Universal Robots URScript: DAS428_958_02_MAR_21_DAS_lado_izquierdo_jig2.script

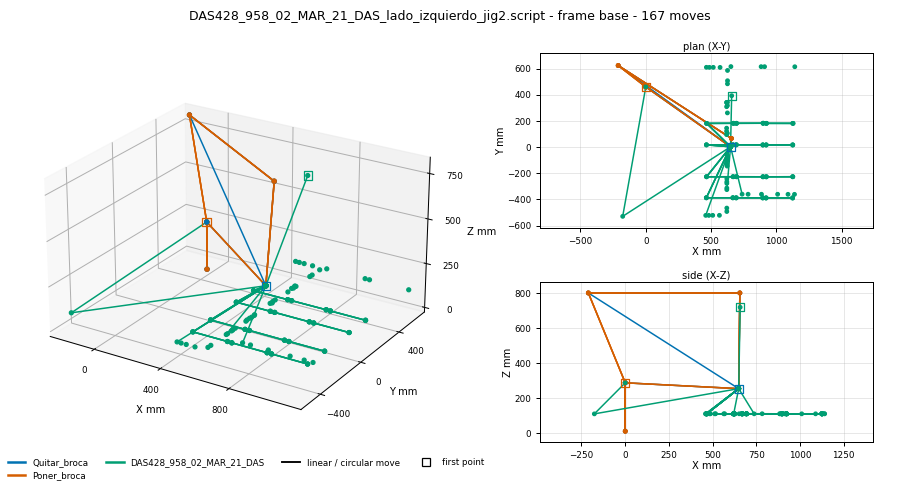
[picture p0: tool path of DAS428_958_02_MAR_21_DAS_lado_izquierdo_jig2.script in frame base, 167 of 755 moves have a stored position in this frame; points joined in program order, loops and branches not executed]
def DAS428_958_02_MAR_21_DAS_lado_izquierdo_jig2():
  step_count_cb486e1e_2b8d_495c_afa4_48e8c6bfd957 = 0
  thread Step_Counter_Thread_418e8cb4_311f_44ce_a52e_b6628405cc57():
    while (True):
      step_count_cb486e1e_2b8d_495c_afa4_48e8c6bfd957 = step_count_cb486e1e_2b8d_495c_afa4_48e8c6bfd957 + 1
      sync()
    end
  end
  run Step_Counter_Thread_418e8cb4_311f_44ce_a52e_b6628405cc57()
  set_safety_mode_transition_hardness(1)
  set_tcp(p[4.109330471764039E-4,-0.21829828276152607,0.037994196120996,1.5580092985761962,-0.12546870791316503,0.12120248426608284])
  set_payload(1.5)
  modbus_add_signal("192.168.10.45", 255, 187, 1, "postrnas_m187", False)
  modbus_set_signal_update_frequency("postrnas_m187", 10)
  modbus_add_signal("192.168.10.45", 255, 289, 1, "ini_cambro_m289", False)
  modbus_set_signal_update_frequency("ini_cambro_m289", 10)
  modbus_add_signal("192.168.10.45", 255, 290, 0, "fin_cambro_m290", False)
  modbus_set_signal_update_frequency("fin_cambro_m290", 10)
  modbus_add_signal("192.168.10.45", 255, 291, 1, "outputbroc_m291", False)
  modbus_set_signal_update_frequency("outputbroc_m291", 10)
  modbus_add_signal("192.168.10.45", 255, 292, 0, "fciclocarr_m292", False)
  modbus_set_signal_update_frequency("fciclocarr_m292", 10)
  modbus_add_signal("192.168.10.45", 255, 7, 1, "avancarrusel_m7", False)
  modbus_set_signal_update_frequency("avancarrusel_m7", 10)
  modbus_add_signal("192.168.10.45", 255, 252, 1, "pose2_m252", False)
  modbus_set_signal_update_frequency("pose2_m252", 10)
  modbus_add_signal("192.168.10.45", 255, 253, 1, "pose3_m253", False)
  modbus_set_signal_update_frequency("pose3_m253", 10)
  modbus_add_signal("192.168.10.45", 255, 254, 1, "pose4_m254", False)
  modbus_set_signal_update_frequency("pose4_m254", 10)
  modbus_add_signal("192.168.10.45", 255, 441, 1, "finciclo_m441", False)
  modbus_set_signal_update_frequency("finciclo_m441", 10)
  modbus_add_signal("192.168.10.45", 255, 442, 1, "finciclo_m442", False)
  modbus_set_signal_update_frequency("finciclo_m442", 10)
  modbus_add_signal("192.168.10.45", 255, 443, 1, "finciclo_m443", False)
  modbus_set_signal_update_frequency("finciclo_m443", 10)
  modbus_add_signal("192.168.10.45", 255, 503, 0, "homecobot_m503", False)
  modbus_set_signal_update_frequency("homecobot_m503", 10)
  modbus_add_signal("192.168.10.45", 255, 288, 1, "cargar_run_m288", False)
  modbus_set_signal_update_frequency("cargar_run_m288", 10)
  modbus_add_signal("192.168.10.45", 255, 287, 0, "desactiver_m288", False)
  modbus_set_signal_update_frequency("desactiver_m288", 10)
  modbus_add_signal("192.168.10.45", 255, 183, 0, "eje7home_m183", False)
  modbus_set_signal_update_frequency("eje7home_m183", 10)
  modbus_add_signal("192.168.10.45", 255, 444, 1, "finciclo_m444", False)
  modbus_set_signal_update_frequency("finciclo_m444", 10)
  modbus_add_signal("192.168.10.45", 255, 381, 0, "pat1_m381", False)
  modbus_set_signal_update_frequency("pat1_m381", 10)
  modbus_add_signal("192.168.10.45", 255, 382, 0, "pat2_m382", False)
  modbus_set_signal_update_frequency("pat2_m382", 10)
  modbus_add_signal("192.168.10.45", 255, 383, 0, "pat3_m383", False)
  modbus_set_signal_update_frequency("pat3_m383", 10)
  modbus_add_signal("192.168.10.45", 255, 384, 0, "pat4_m384", False)
  modbus_set_signal_update_frequency("pat4_m384", 10)
  modbus_add_signal("192.168.10.45", 255, 385, 0, "pat5_m385", False)
  modbus_set_signal_update_frequency("pat5_m385", 10)
  modbus_add_signal("192.168.10.45", 255, 386, 0, "pat6_m386", False)
  modbus_set_signal_update_frequency("pat6_m386", 10)
  modbus_add_signal("192.168.10.45", 255, 387, 0, "pat7_m387", False)
  modbus_set_signal_update_frequency("pat7_m387", 10)
  modbus_add_signal("192.168.10.45", 255, 388, 0, "pat8_m388", False)
  modbus_set_signal_update_frequency("pat8_m388", 10)
  modbus_add_signal("192.168.10.45", 255, 389, 0, "pat9_m389", False)
  modbus_set_signal_update_frequency("pat9_m389", 10)
  modbus_add_signal("192.168.10.45", 255, 390, 0, "pat10_m390", False)
  modbus_set_signal_update_frequency("pat10_m390", 10)
  modbus_add_signal("192.168.10.45", 255, 391, 0, "pat11_m391", False)
  modbus_set_signal_update_frequency("pat11_m391", 10)
  modbus_add_signal("192.168.10.45", 255, 392, 0, "pat12_m392", False)
  modbus_set_signal_update_frequency("pat12_m392", 10)
  modbus_add_signal("192.168.10.45", 255, 401, 0, "inipat1_m401", False)
  modbus_set_signal_update_frequency("inipat1_m401", 10)
  modbus_add_signal("192.168.10.45", 255, 402, 0, "inipat2_m402", False)
  modbus_set_signal_update_frequency("inipat2_m402", 10)
  modbus_add_signal("192.168.10.45", 255, 403, 0, "inipat3_m403", False)
  modbus_set_signal_update_frequency("inipat3_m403", 10)
  modbus_add_signal("192.168.10.45", 255, 404, 0, "inipat4_m404", False)
  modbus_set_signal_update_frequency("inipat4_m404", 10)
  modbus_add_signal("192.168.10.45", 255, 405, 0, "inipat5_m405", False)
  modbus_set_signal_update_frequency("inipat5_m405", 10)
  modbus_add_signal("192.168.10.45", 255, 406, 0, "inipat6_m406", False)
  modbus_set_signal_update_frequency("inipat6_m406", 10)
  modbus_add_signal("192.168.10.45", 255, 407, 0, "inipat7_m407", False)
  modbus_set_signal_update_frequency("inipat7_m407", 10)
  modbus_add_signal("192.168.10.45", 255, 408, 0, "inipat8_m408", False)
  modbus_set_signal_update_frequency("inipat8_m408", 10)
  modbus_add_signal("192.168.10.45", 255, 409, 0, "inipat9_m409", False)
  modbus_set_signal_update_frequency("inipat9_m409", 10)
  modbus_add_signal("192.168.10.45", 255, 410, 0, "inipat10_m410", False)
  modbus_set_signal_update_frequency("inipat10_m410", 10)
  modbus_add_signal("192.168.10.45", 255, 411, 0, "inipat11_m411", False)
  modbus_set_signal_update_frequency("inipat11_m411", 10)
  modbus_add_signal("192.168.10.45", 255, 412, 0, "inipat12_m412", False)
  modbus_set_signal_update_frequency("inipat12_m412", 10)
  modbus_add_signal("192.168.10.45", 255, 430, 0, "modeloDer_m430", False)
  modbus_set_signal_update_frequency("modeloDer_m430", 10)
  modbus_add_signal("192.168.10.45", 255, 380, 1, "mensaje_m380", False)
  modbus_set_signal_update_frequency("mensaje_m380", 10)
  modbus_add_signal("192.168.10.45", 255, 379, 0, "respues_m379", False)
  modbus_set_signal_update_frequency("respues_m379", 10)
  modbus_add_signal("192.168.10.45", 255, 251, 1, "pose1_m251", False)
  modbus_set_signal_update_frequency("pose1_m251", 10)
  modbus_set_runstate_dependent_choice("postrnas_m187",0)
  modbus_set_runstate_dependent_choice("ini_cambro_m289",0)
  modbus_set_runstate_dependent_choice("outputbroc_m291",0)
  modbus_set_runstate_dependent_choice("avancarrusel_m7",0)
  modbus_set_runstate_dependent_choice("pose2_m252",0)
  modbus_set_runstate_dependent_choice("pose3_m253",0)
  modbus_set_runstate_dependent_choice("pose4_m254",0)
  modbus_set_runstate_dependent_choice("finciclo_m441",0)
  modbus_set_runstate_dependent_choice("finciclo_m442",0)
  modbus_set_runstate_dependent_choice("finciclo_m443",0)
  modbus_set_runstate_dependent_choice("cargar_run_m288",0)
  modbus_set_runstate_dependent_choice("finciclo_m444",0)
  modbus_set_runstate_dependent_choice("mensaje_m380",0)
  modbus_set_runstate_dependent_choice("pose1_m251",0)
  set_standard_analog_input_domain(0, 1)
  set_standard_analog_input_domain(1, 1)
  set_tool_analog_input_domain(0, 1)
  set_tool_analog_input_domain(1, 1)
  set_analog_outputdomain(0, 0)
  set_analog_outputdomain(1, 0)
  set_input_actions_to_default()
  set_runstate_standard_digital_outputs([2])
  set_runstate_configurable_digital_outputs([1])
  set_runstate_standard_digital_output_to_value(2, 1)
  set_runstate_configurable_digital_output_to_value(1, 1)
  set_gravity([0.0, 0.0, 9.82])
  set_tool_communication(False, 115200, 0, 1, 1.5, 3.5)
  set_tool_output_mode(0)
  set_tool_digital_output_mode(0, 1)
  set_tool_digital_output_mode(1, 1)
  set_tool_voltage(0)
  global contador=0
  global i_var_1=0
  global Pallet_1_cnt_1=1
  global Pallet_1_cnt=1
  global Line_1=p[0.0,0.0,0.0,0.0,0.0,0.0]
  global Line_2=p[0.0,0.0,0.0,0.0,0.0,0.0]
  global Line_3=p[0.0,0.0,0.0,0.0,0.0,0.0]
  global Line_4=p[-0.2932874787951964,0.3932288129452105,0.013749459185886714,0.019478391032120013,-0.0350876085014595,1.5300278925331599]
  global Line_5=p[0.0,0.0,0.0,0.0,0.0,0.0]
  global Plane_1=p[-0.4357649673792705,0.3571224276764373,-0.011331751409534768,-0.03455953496512708,-0.012487423981114925,3.103751116092306]
  global Plane_2=p[-0.4823864034329737,0.3302516442079689,0.014283714098506706,0.017125077458443067,0.05770060098903715,-2.9134709732588786]
  global Plane_3=p[0.003678615545088639,0.4082921331082374,0.10477407557236007,-2.072177303174012E-4,7.379081343290108E-4,-6.424400645467977E-4]
  global Plane_4=p[-0.4500206307677429,-0.2823718146925442,-0.4767416657426552,0.013278190059218174,0.013334473770785706,1.8479691991032237]
  global Plano_patron1=p[-0.7699005610122596,0.304894434078545,0.0420369514744936,-0.0031270356010209216,1.7180543614697593E-4,-3.508888786211572E-5]
  global Point_13=p[0.0,0.0,0.0,0.0,0.0,0.0]
  global Point_3=p[0.0,0.0,0.0,0.0,0.0,0.0]
  global Point_8=p[0.0,0.0,0.0,0.0,0.0,0.0]
  global Punto_prot_1=p[0.0,0.0,0.0,0.0,0.0,0.0]
  global Punto_seg_der=p[0.23741638234469645,0.3587772222537799,0.42419077585740217,0.818517054876345,1.4216436941132238,1.005041187710707]
  global pisp_958=p[-0.41395442210486977,-0.2082168853247176,0.041553466664982,0.014014788518713659,0.01101911827984854,1.569193423241601]
  rtde_set_watchdog("speed_slider_mask", 10.0, "ignore")
  global Traslacion_p=p[.657998712498, .394119076430, .719668538659, .745859698144, 2.906519637838, .095468097993]
  global Traslacion_q=[-3.020863008919047, -1.4521287285823696, 0.9893999609737083, 0.3161356049923509, -5.817383157179211, 7.125860208047008E-4]
  global Home2_p=p[.649602302195, .003200282484, .254149874925, -2.448457879294, -1.966199736652, -.011076409707]
  global Home2_q=[-3.47968947108801, -1.6856169348881274, 2.036329601799979, -0.3455951480915882, -4.992365550646321, 0.0060764790449239214]
  global Home3_p=p[.649602302195, .003200282484, .254149874925, -2.448457879294, -1.966199736652, -.011076409707]
  global Home3_q=[-3.479689471087993, -1.6856169348881211, 2.0363296017999737, -0.34559514809159, -4.992365550646304, 0.006076479044924019]
  global Home4_p=p[.649602302195, .003200282484, .254149874925, -2.448457879294, -1.966199736652, -.011076409707]
  global Home4_q=[-3.479689471087993, -1.6856169348881211, 2.0363296017999737, -0.34559514809159, -4.992365550646304, 0.006076479044924019]
  global PosicionApagado_p=p[-.175961014487, -.529389253007, .109949884724, .175001600804, 2.113291246609, -2.157399109703]
  global PosicionApagado_q=[-1.5727354621284952, -1.5704867605983486, -2.807039864148308, -0.30557696332673245, -4.706711136129834, 1.778107977035495E-5]
  global Precambio_broca_p=p[.000830370305, .461517540512, .287521124194, -.221784750204, -3.131955254916, .000429460883]
  global Precambio_broca_q=[-2.1838225298159477, -2.0964618902985066, 2.243453456263678, -0.13436505871461257, -5.342774534909408, -0.004043449473680738]
  global Linea1_A_p=p[.465780239716, -.226284822275, .110110305320, 3.129199777247, .273979671894, -.008474561279]
  global Linea1_A_q=[-3.7622293747396913, -1.6873556925995992, 2.323362421011069, -0.625104012809361, -4.0968533396839515, 0.0033473062041684543]
  global Linea1_B_p=p[.669199999133, -.226066231601, .110221514703, 3.129199488643, .274057096186, -.008522317905]
  global Linea1_B_q=[-3.557231781452517, -1.3492008498278363, 1.961545229349972, -0.5993084840575982, -3.891978745553196, 0.0068914536813957416]
  global Linea1_C_p=p[.694599999674, -.226083076366, .110775282131, 3.129206209142, .274048762949, -.008557115599]
  global Linea1_C_q=[-3.5408294989047437, -1.3120520197143488, 1.9116878668393618, -0.5863558735051146, -3.8755559725861075, 0.007215554028316085]
  global Linea1_D_p=p[.897799999597, -.226330598752, .110549197198, 3.129164560911, .274100632214, -.008493112790]
  global Linea1_D_q=[-3.4452506974721455, -1.015094527261077, 1.4697422225132426, -0.4398923161705586, -3.779757131526884, 0.009316440733303288]
  global Linea1_E_p=p[.923199997743, -.226496087218, .110278761023, 3.129196935269, .274071665669, -.008639622731]
  global Linea1_E_q=[-3.436588597727809, -0.976349509057826, 1.4065148117166615, -0.4151627604596042, -3.7710218003171097, 0.009513196103198673]
  global Linea1_F_p=p[1.125593354651, -.226031138561, .110601831768, 3.129192254502, .274074519951, -.008696700454]
  global Linea1_F_q=[-3.380697676481182, -0.6099111929302072, 0.7528298757650722, -0.1267902515679964, -3.714400713814072, 0.010912064972982147]
  def calculate_point_to_move_towards(feature, direction, position_distance):
    local posDir=[direction[0], direction[1], direction[2]]
    if (norm(posDir) < 1e-6):
      return get_target_waypoint()
    end
    local direction_vector_normalized=normalize(posDir)
    local displacement_pose=p[direction_vector_normalized[0] * position_distance,direction_vector_normalized[1] * position_distance,direction_vector_normalized[2] * position_distance,0,0,0]
    local wanted_displacement_in_base_frame=pose_sub(pose_trans(feature, displacement_pose), feature)
    return pose_add(get_target_waypoint(), wanted_displacement_in_base_frame)
  end
  global Linea2_A_p=p[.466954168710, .182156727796, .110171699464, -2.448457838983, -1.966199888042, -.011076390033]
  global Linea2_A_q=[-3.096264362332022, -1.8105063261906196, 2.419381749575411, -0.604569943120544, -4.609367858418758, 0.008210447251383535]
  global Linea2_B_p=p[.671809999536, .182878038708, .110175282179, -2.448398718020, -1.966214966670, -.010953917198]
  global Linea2_B_q=[-3.112193266343249, -1.4618930385561022, 2.1005475692711357, -0.6342202128720773, -4.625507134533515, 0.00845567105716949]
  global Linea2_C_p=p[.694980620228, .182769618296, .110459932861, -2.448327792652, -1.966241960778, -.010898882344]
  global Linea2_C_q=[-3.1136170783763246, -1.427697328825201, 2.059986020915073, -0.6277999413035573, -4.626970277725095, 0.008475304624878617]
  global Linea2_D_p=p[.898787430028, .183234989861, .110403286316, -2.448304893977, -1.966353718915, -.010975641562]
  global Linea2_D_q=[-3.12042574519119, -1.1376151787135544, 1.6647315225706083, -0.5226894752077342, -4.633689721395611, 0.008491290355203619]
  global Linea2_E_p=p[.923789841802, .182506729307, .110323521287, -2.448339335785, -1.966352412105, -.011034134800]
  global Linea2_E_q=[-3.1220303350773233, -1.1024169697310633, 1.610792612077442, -0.5039930836645397, -4.635244042411777, 0.008484609097352974]
  global Linea2_F_p=p[1.126945944045, .182371421241, .110084235246, -2.448292218177, -1.966366471653, -.011020014588]
  global Linea2_F_q=[-3.126205891145389, -0.7888654762746627, 1.0844527378197477, -0.2911805586510319, -4.6389576225939395, 0.008426573530911268]
  global Linea7_A_p=p[.737913382913, -.359696656416, .110246852616, 3.131872092311, .186635383423, -.000389334829]
  global Linea7_A_q=[-3.681156562266171, -1.1996168071622932, 1.757330151202673, -0.5522026597660465, -3.9601640674441323, 0.005316316519943243]
  global Linea7_B_p=p[.783713148217, -.360080715325, .110620974020, 3.131872080694, .186635404395, -.000389343545]
  global Linea7_B_q=[-3.650143104990655, -1.1359413316685298, 1.6616529669860118, -0.5200665751996176, -3.929093763815281, 0.005555397450602444]
  global Linea8_A_p=p[.886282799932, -.360229310841, .110453772921, 3.131519956407, .186494776915, .000579777937]
  global Linea8_A_q=[-3.591304287493482, -0.9891617182428476, 1.4289624761138866, -0.4346002764061705, -3.870006358141346, 0.006011745682200086]
  global Linea8_B_p=p[1.009987450255, -.360229310302, .110179227584, 3.131519925151, .186494817820, .000579759973]
  global Linea8_B_q=[-3.5358660704998717, -0.7924298121308935, 1.0907006839592273, -0.2928265782260997, -3.8142305776877343, 0.0064076248760271785]
  global Linea9_A_p=p[1.089313325367, -.360630550626, .110237381886, 3.131274831042, .186572958872, .001401500331]
  global Linea9_A_q=[-3.507282006423159, -0.6385942191612735, 0.8089501351297868, -0.1653539889318978, -3.785363860326909, 0.006616479785108709]
  global Linea9_B_p=p[1.138944388844, -.360869351507, .110826017632, 3.131274802661, .186572988174, .001401483023]
  global Linea9_B_q=[-3.4914339632991864, -0.5124624399707418, 0.5676507222077732, -0.05011131989687101, -3.7691835676211607, 0.006732071657192494]
  global Linea10_A_p=p[.620978322043, -.324892456797, .110623766440, 3.127402623628, -.245143091263, -.004063554207]
  global Linea10_A_q=[-3.6869382053447044, -1.3223584773988293, 1.927375204305715, -0.5983630349819116, -3.6905142249820324, 0.0056231827538635315]
  global Linea10_B_p=p[.621097917225, -.276980216964, .110320290981, 3.127402605879, -.245143081258, -.004063559866]
  global Linea10_B_q=[-3.6188087722380935, -1.3384072237024949, 1.949063614559142, -0.6032315503323895, -3.6223937108691318, 0.006590396406481958]
  global Linea11_A_p=p[.623455356385, -.144672989900, .110191487849, -2.632012907887, -1.710466693368, -.008551801775]
  global Linea11_A_q=[-3.7294766647125748, -1.5700524659119814, 2.21580175367518, -0.6379282889546607, -5.042121691434226, 0.005581533742989642]
  global Linea11_B_p=p[.624119671393, -.090095469021, .110353884155, -2.632012896780, -1.710466734062, -.008551794970]
  global Linea11_B_q=[-3.6247502966617073, -1.585150048761757, 2.2304099707796063, -0.6377871669514974, -4.937393005511421, 0.006400309223622675]
  global Linea12_A_p=p[.624141411120, -.066274166300, .110334660294, -2.632061457031, -1.710628419892, -.008680091079]
  global Linea12_A_q=[-3.576867818672329, -1.5888248455929554, 2.23409769230859, -0.638081681915871, -4.88958008805711, 0.006759858484637715]
  global Linea12_B_p=p[.625005135416, .106664404916, .110180545519, -2.632061469151, -1.710628482598, -.008680127081]
  global Linea12_B_q=[-3.2068887547507323, -1.551909790420524, 2.1974871560020848, -0.638805025446775, -4.519623607927026, 0.009359012311380255]
  global Linea13_A_p=p[.625493298354, .262478777538, .110355483985, -2.632548083396, -1.710921113652, -.010070841951]
  global Linea13_A_q=[-2.896364151370071, -1.4448052024132805, 2.0799552622917368, -0.6290694071523859, -4.209104057924403, 0.011452105368751556]
  global Linea13_B_p=p[.625493296860, .318856578939, .110131630173, -2.632548086986, -1.710921163442, -.010070846484]
  global Linea13_B_q=[-2.7987199569733097, -1.394849229494266, 2.020507255629248, -0.6192929302058419, -4.111456896339345, 0.012194173917594142]
  global Linea14_A_p=p[.625748762392, .343504937265, .110090990642, -2.632595117185, -1.711060508708, -.011002715073]
  global Linea14_A_q=[-2.7589776121724974, -1.371725061704466, 1.991938508379024, -0.614306407879349, -4.0717686455064666, 0.012519321582973785]
  global Linea14_B_p=p[.626022539964, .485152545421, .110593753972, -2.632595124419, -1.711060553733, -.011002727305]
  global Linea14_B_q=[-2.561324434207597, -1.228184115147677, 1.79766140697026, -0.5625917279677406, -3.874049521809336, 0.014268843198803616]
  global Linea15_A_p=p[.626306650398, .508674603028, .110445455669, -2.632595127775, -1.711060613121, -.011002737975]
  global Linea15_A_q=[-2.533508862703878, -1.202261171286347, 1.7605999966793635, -0.55125669711577, -3.846216171124823, 0.014567785906905393]
  global Linea15_B_p=p[.626327608491, .587415564298, .110050045410, -2.632661246672, -1.711049389617, -.010999857798]
  global Linea15_B_q=[-2.4482942280068585, -1.1131828351876312, 1.6277564152308788, -0.5068229975694187, -3.760894753760676, 0.015518000293985423]
  global Linea16_A_p=p[.464714302335, .611413139504, .110697464349, -1.544268383540, -2.732104823202, -.006884184964]
  global Linea16_A_q=[-2.4550359831168613, -1.3587121352385232, 1.9739909556549193, -0.6095013542703764, -4.727784672200272, 0.006868741264362654]
  global Linea16_B_p=p[.487741348141, .611017673565, .110415464036, -1.544268358835, -2.732104854917, -.006884177480]
  global Linea16_B_q=[-2.4794279049425754, -1.3389262434910556, 1.9490984118290324, -0.604365353535707, -4.75217062245783, 0.006734800587170575]
  global Linea17_A_p=p[.517383659268, .611103429132, .110729179233, -1.544779713402, -2.732685367780, -.009945500495]
  global Linea17_A_q=[-2.5082575279683113, -1.3131453182243042, 1.9151753969774692, -0.598283135183288, -4.78088650060061, 0.00668272054728547]
  global Linea17_B_p=p[.569253413106, .610696887479, .110460451666, -1.544779672167, -2.732685417131, -.009945491911]
  global Linea17_B_q=[-2.5549019817458243, -1.2642731579102362, 1.8492778264267276, -0.5811941707445918, -4.827506542897114, 0.006516537786687767]
  global Linea18_A_p=p[.652275282871, .616966070789, .110402012202, -1.544268371887, -2.732104838867, -.006884188160]
  global Linea18_A_q=[-2.6106362750002035, -1.1730578134725853, 1.7176129055392177, -0.5385325271143078, -4.883275143872667, 0.005979356975084116]
  global Linea18_AB_p=p[.883614943259, .616349563116, .110351134256, -1.544268345639, -2.732104870876, -.006884192709]
  global Linea18_AB_q=[-2.7386992398245744, -0.9017900558849279, 1.281606576558123, -0.3734626609773617, -5.010988146234565, 0.005130637771908034]
  global Linea18_BA_p=p[.909904961943, .616222280799, .110421447666, -1.544268322161, -2.732104902209, -.006884182125]
  global Linea18_BA_q=[-2.7498726987223208, -0.8660697617883866, 1.2197485096371476, -0.3472882558118906, -5.02209865790525, 0.005047885057257062]
  global Linea18_B_p=p[1.141235285063, .615792039333, .110307833561, -1.544268303833, -2.732104945128, -.006884144817]
  global Linea18_B_q=[-2.8277732907081354, -0.39061700846990277, 0.32871463965525227, 0.06857809871196263, -5.098826528836324, 0.004459377539679431]
  global Linea3_A_p=p[.464230833806, -.387159783178, .110302837424, -2.419116994491, -2.002063214725, -.010924024823]
  global Linea3_A_q=[-4.3910163833731914, -1.555782586510814, 2.202005657326122, -0.6299721466298944, -5.933748291401908, -0.006546668033756475]
  global Linea3_B_p=p[.667429999599, -.387164709724, .110463996486, -2.419112960004, -2.002099447112, -.010918294544]
  global Linea3_B_q=[-4.057680660838788, -1.323350209478841, 1.9290195916743436, -0.5973157418827517, -5.6004464441758355, 0.0019643644184652587]
  global Linea3_C_p=p[.692830001733, -.387650681328, .110109359717, -2.419059878647, -2.002159205155, -.010925286677]
  global Linea3_C_q=[-4.026535686604552, -1.2922202748569482, 1.8881224565782944, -0.5878969018347195, -5.569340867091353, 0.002380584369406691]
  global Linea3_D_p=p[.896029998777, -.387852804805, .110196889251, -2.419080439535, -2.002173420011, -.010934520449]
  global Linea3_D_q=[-3.829265965876175, -1.0382006055234712, 1.5094078253308432, -0.4647896797065121, -5.371850161314754, 0.004346050949126656]
  global Linea3_E_p=p[.921429998459, -.388319341203, .110580746835, -2.419087749766, -2.002201874505, -.010952866993]
  global Linea3_E_q=[-3.8105196931013556, -1.0042069202420114, 1.4534307338800188, -0.442942131267305, -5.3530686968067505, 0.004496004728317427]
  global Linea3_F_p=p[1.124629998567, -.388399736062, .110402465879, -2.419125348681, -2.002211693637, -.010968628578]
  global Linea3_F_q=[-3.686825535686765, -0.6866169613755719, 0.8978925546882044, -0.20560612623027819, -5.228777140850181, 0.005303851178450003]
  global Linea4_A_p=p[.464979976316, .017836773167, .110310404991, -2.448457836899, -1.966199895061, -.011076466632]
  global Linea4_A_q=[-3.6529867765693265, -1.9452905946133079, 2.501674762544585, -0.5506678388692903, -5.165918169719263, 0.005229115013293928]
  global Linea4_B_p=p[.668170000037, .017833792943, .110301370691, -2.448481013042, -1.966150615318, -.011068565459]
  global Linea4_B_q=[-3.4381583087354946, -1.5218818556667548, 2.1666255386489652, -0.6398943768365513, -4.9513971286391545, 0.00694330599646038]
  global Linea4_C_p=p[.693569999371, .018136934193, .110396766029, -2.448555603805, -1.966143161170, -.011081417994]
  global Linea4_C_q=[-3.4230261654246217, -1.4801703680484923, 2.12081541771418, -0.6358791842300828, -4.9362363497913835, 0.007021482749777874]
  global Linea4_D_p=p[.896769999275, .017310642274, .110305174457, -2.448571849199, -1.966119022896, -.011066680754]
  global Linea4_D_q=[-3.3451971602477997, -1.174492939736922, 1.7203661334209173, -0.541265722112624, -4.858269381434981, 0.007475731853766376]
  global Linea4_E_p=p[.922169999701, .017310244028, .110356528892, -2.448641417951, -1.966134840023, -.011114602385]
  global Linea4_E_q=[-3.338321082289934, -1.1376526551075221, 1.6649290062563085, -0.5227466706314932, -4.8513393849974475, 0.0074892124034669355]
  global Linea4_F_p=p[1.125369999206, .017258611272, .110276213649, -2.448642075535, -1.966106276713, -.011053663852]
  global Linea4_F_q=[-3.296678674914709, -0.823269689152891, 1.1453259230712316, -0.31754572368232736, -4.809226384426388, 0.007609882209201224]
  global Linea19_A_p=p[.459500483192, -.521966359264, .110287307573, 2.444310209774, 1.962895565264, .013982840383]
  global Linea19_A_q=[-4.471273749261577, -1.392054727345812, 2.0194079671963188, -0.631880630087049, -5.984536630474428, 0.008512064870961566]
  global Linea19_B_p=p[.483360000235, -.521950949871, .110282315610, 2.444325023128, 1.962902223119, .013994776933]
  global Linea19_B_q=[-4.431418332577646, -1.3728259473858282, 1.9954261647225349, -0.6266575038166051, -5.944674315997971, 0.007991292980141475]
  global Linea20_A_p=p[.513036034860, -.521545431794, .110268231563, 2.444009364395, 1.962577422245, .013682365965]
  global Linea20_A_q=[-4.3834965789724585, -1.3484805306961114, 1.9644732931448647, -0.6200502308609375, -5.896708193899019, 0.007411715416055564]
  global Linea20_B_p=p[.564367225862, -.521477319483, .110373765560, 2.444016038345, 1.962504003089, .013643134348]
  global Linea20_B_q=[-4.3058887078080375, -1.3027271523559243, 1.9039833103281723, -0.6047911467897613, -5.819042462186221, 0.0066992366938736225]
  global Linea22_A_p=p[.620834960282, -.492247478559, .110497141865, 2.443672554456, 1.961786926726, .013351573251]
  global Linea22_A_q=[-4.206755740765137, -1.2804659183319655, 1.8736182491376765, -0.5968641932902443, -5.719676086958917, 0.005935095196567525]
  global Linea22_B_p=p[.620833404792, -.466079999734, .110459690156, 2.443722512690, 1.961793090207, .013354519254]
  global Linea22_B_q=[-4.1866126282627825, -1.3077962244491328, 1.9107030191507974, -0.6064669786035877, -5.699529941145465, 0.005780495013403351]
  global Linea23_A_p=p[.621024526563, -.312761557524, .110089939756, 2.443246126125, 1.961395760010, .013163762842]
  global Linea23_A_q=[-4.036926680747516, -1.4547656269869815, 2.0950717331465434, -0.6438091569554754, -5.5498710282044215, 0.004712934754347309]
  global Linea23_B_p=p[.621018358815, -.264150000183, .110084555763, 2.443270526968, 1.961384280882, .013190437581]
  global Linea23_B_q=[-3.9759151346568355, -1.4950906707753084, 2.140588135264717, -0.6488316844199273, -5.488842649275668, 0.0044022199091813975]
  global Linea24_A_p=p[.621098439622, -.240775675200, .110574395502, 2.442915738284, 1.960990434209, .013229551219]
  global Linea24_A_q=[-3.943688610074833, -1.5136152224729447, 2.1598199021528064, -0.6499650281649636, -5.456556883931132, 0.004208571162668064]
  global Linea24_B_p=p[.621118179566, -.130050000223, .110593596533, 2.442940887576, 1.960970321451, .013243383298]
  global Linea24_B_q=[-3.7657146588007127, -1.5803190255179214, 2.228636133114988, -0.6517531716906797, -5.2785469770071005, 0.0033512703841079025]
  global Linea25_A_p=p[.621437015783, -.106982911313, .110365967551, 2.442654836858, 1.960739689231, .013433900484]
  global Linea25_A_q=[-3.7228620416933285, -1.5889924294860043, 2.2377643530667757, -0.6525555528636033, -5.235691478214098, 0.0031786304463132424]
  global Linea25_B_p=p[.621448492153, -.058220000048, .110378145190, 2.442603922060, 1.960750387302, .013453779592]
  global Linea25_B_q=[-3.6275781962436264, -1.6026393687452547, 2.2509404516858775, -0.6520428035114243, -5.140428502414784, 0.0027627020952146345]
  global Linea26_A_p=p[.619159227850, .096338884870, .110740941987, .899978624169, 3.001630062312, .019199733645]
  global Linea26_A_q=[-3.5390754743527815, -1.4787706815615067, 2.123788189423017, -0.778642028497547, -6.257990636071562, 0.1308097629133993]
  global Linea26_B_p=p[.619176001176, .121859999719, .110738192265, .900005863428, 3.001632041634, .019205064751]
  global Linea26_B_q=[-3.4941546104866616, -1.4665413577991107, 2.1079108634834878, -0.6895245612943697, -6.213138821490713, 0.04522556275457999]
  global Linea27_A_p=p[.619470388681, .145721512233, .110285520947, .899984863397, 3.001101158686, .019169741261]
  global Linea27_A_q=[-3.4511962546946826, -1.4630482655533044, 2.104742069163123, -0.6720639641347148, -6.17011399581671, 0.026805913560317585]
  global Linea27_B_p=p[.619467972926, .310059999998, .110284525077, .899976853464, 3.001034446604, .019158185330]
  global Linea27_B_q=[-3.1499341209632474, -1.4192801482839945, 2.053305987085655, -0.6428059491629234, -5.868866145482653, 0.004292910361343351]
  global Linea28_B_p=p[.619758029730, .342258392106, .110153188185, .899916349228, 3.000597837149, .019434917209]
  global Linea28_B_q=[-3.0923901875970277, -1.402935932194037, 2.0338680097589563, -0.6392981617522118, -5.811277262215688, 0.0032495578488829224]
  global Precam_bro1_p=p[.656076269686, .067103652830, .801529194085, 2.333752758408, 2.077660178403, .030474428127]
  global Precam_bro1_q=[-3.3770460833376266, -1.5485738802438487, 0.9024271451168131, 0.6289852346296929, -4.989016163426699, 0.005603611084501629]
  global Precam_bro2_p=p[-.210318050744, .625064228220, .801529194085, .167219476409, -3.132160268904, -.039745099994]
  global Precam_bro2_q=[-1.5836008221808306, -1.5485738802438487, 0.9024271451168131, 0.6289852346296929, -4.989016163426699, 0.005603611084501629]
  global Dejar_broca_p=p[.000823895285, .461515686418, .010824983886, -.221812507768, -3.131977618886, .000372128741]
  global Dejar_broca_q=[-2.183487269545523, -1.7626289818446779, 2.619089631151862, -0.8448915610823917, -5.34389996121201, -0.0023222697552238714]
  def Quitar_broca():
    $ 5334 "Quitar_broca" "noBreak"
    $ 5335 "Quitar_broca"
    $ 5336 "barrenos_hechos≔barrenos_hechos+1"
    global barrenos_hechos=barrenos_hechos+1
    $ 5341 "If barrenos_hechos≟14 or cambiar_broca≟ True "
    if (barrenos_hechos == 14  or  cambiar_broca ==   True  ):
      $ 5342 "'Codigo de quitar broca'"
      # 'Codigo de quitar broca'
      $ 5343 "MoveL"
      $ 5344 "Direction: Base Z+"
      global move_thread_flag_5344=0
      thread move_thread_5344():
        enter_critical
        move_thread_flag_5344 = 1
        local towardsPos=calculate_point_to_move_towards(p[0.0,0.0,0.0,0.0,0.0,0.0], [0.0,0.0,1.0], 0.1)
        movel(towardsPos, a=1.2, v=0.25)
        move_thread_flag_5344 = 2
        exit_critical
      end
      move_thread_flag_5344 = 0
      move_thread_han_5344 = run move_thread_5344()
      while (True):
        sleep(1.0E-10)
        if (move_thread_flag_5344 > 1):
          join move_thread_han_5344
          $ 5345 "Until (distance)"
          break
        end
        sync()
      end
      $ 5346 "If eje7≟3"
      if (eje7 == 3):
        $ 5347 "Home3" "breakAfter"
        movel(Home3_p, a=1.2, v=0.25)
        $ 5348 "Precam_bro1" "breakAfter"
        movel(Precam_bro1_p, a=1.2, v=0.25)
        $ 5349 "Precam_bro2" "breakAfter"
        movel(Precam_bro2_p, a=1.2, v=0.25)
      end
      $ 5350 "If eje7≟2"
      if (eje7 == 2):
        $ 5351 "Home2" "breakAfter"
        movel(Home2_p, a=1.2, v=0.25)
      end
      $ 5353 "Precambio_broca" "breakAfter"
      movel(Precambio_broca_p, a=1.2, v=0.25)
      $ 5354 "Dejar_broca" "breakAfter"
      movel(Dejar_broca_p, a=0.1, v=0.09)
      $ 5355 "Set outputbroc_m291=Encender"
      modbus_set_output_signal("outputbroc_m291", True)
      $ 5356 "Wait: 2.0"
      sleep(2.0)
      $ 5358 "Wait: 2.0"
      sleep(2.0)
      $ 5359 "Set outputbroc_m291=Apagar"
      modbus_set_output_signal("outputbroc_m291", False)
      $ 5360 "Wait: 0.5"
      sleep(0.5)
      $ 5361 "Wait fciclocarr_m292=LO"
      while (modbus_get_signal_status("fciclocarr_m292") == True):
        sync()
      end
      $ 5362 "Wait: 0.5"
      sleep(0.5)
      $ 5364 "MoveL"
      $ 5365 "Precambio_broca" "breakAfter"
      movel(Precambio_broca_p, a=0.1, v=0.09)
      $ 5366 "Set avancarrusel_m7=Encender"
      modbus_set_output_signal("avancarrusel_m7", True)
      $ 5367 "Wait: 1.0"
      sleep(1.0)
      $ 5368 "Wait: 0.1"
      sleep(0.1)
    end
  end
  def Poner_broca():
    $ 5369 "Poner_broca" "noBreak"
    $ 5370 "Poner_broca"
    $ 5371 "If cambiar_broca≟ True  or iniciando_prog≟ True "
    if (cambiar_broca ==   True    or  iniciando_prog ==   True  ):
      $ 5372 "'Codigo de poner broca'"
      # 'Codigo de poner broca'
      $ 5373 "Set ini_cambro_m289=Apagar"
      modbus_set_output_signal("ini_cambro_m289", False)
      $ 5374 "MoveL"
      $ 5375 "Precambio_broca" "breakAfter"
      movel(Precambio_broca_p, a=1.2, v=0.25)
      $ 5376 "Popup: Cambia a las siguientes brocas"
      popup("Cambia a las siguientes brocas", "Advertencia", True, False, blocking=True)
      $ 5377 "Dejar_broca" "breakAfter"
      movel(Dejar_broca_p, a=0.1, v=0.09)
      $ 5378 "Set ini_cambro_m289=Encender"
      modbus_set_output_signal("ini_cambro_m289", True)
      $ 5379 "Wait: 2.0"
      sleep(2.0)
      $ 5381 "Wait: 2.0"
      sleep(2.0)
      $ 5382 "Set ini_cambro_m289=Apagar"
      modbus_set_output_signal("ini_cambro_m289", False)
      $ 5383 "Wait: 0.5"
      sleep(0.5)
      $ 5384 "Wait fciclocarr_m292=LO"
      while (modbus_get_signal_status("fciclocarr_m292") == True):
        sync()
      end
      $ 5385 "Wait: 0.5"
      sleep(0.5)
      $ 5387 "MoveL"
      $ 5388 "Precambio_broca" "breakAfter"
      movel(Precambio_broca_p, a=0.1, v=0.09)
      $ 5389 "If eje7≟3"
      if (eje7 == 3):
        $ 5390 "Precam_bro2" "breakAfter"
        movel(Precam_bro2_p, a=1.2, v=0.25)
        $ 5391 "Precam_bro1" "breakAfter"
        movel(Precam_bro1_p, a=1.2, v=0.25)
        $ 5392 "Home3" "breakAfter"
        movel(Home3_p, a=1.2, v=0.25)
      end
      $ 5393 "If eje7≟2"
      if (eje7 == 2):
        $ 5395 "Home2" "breakAfter"
        movel(Home2_p, a=1.2, v=0.25)
      end
      $ 5396 "barrenos_hechos≔0"
      global barrenos_hechos=0
      $ 5397 "iniciando_prog≔ False "
      global iniciando_prog=  False
      $ 5398 "cambiar_broca≔ False "
      global cambiar_broca=  False
    end
    $ 5399 "If barrenos_hechos≟14"
    if (barrenos_hechos == 14):
      $ 5400 "If cambiar_broca≟ False "
      if (cambiar_broca ==   False  ):
        $ 5401 "'Codigo de poner broca'"
        # 'Codigo de poner broca'
        $ 5402 "Set ini_cambro_m289=Apagar"
        modbus_set_output_signal("ini_cambro_m289", False)
        $ 5403 "MoveL"
        $ 5404 "Precambio_broca" "breakAfter"
        movel(Precambio_broca_p, a=1.2, v=0.25)
        $ 5405 "Dejar_broca" "breakAfter"
        movel(Dejar_broca_p, a=0.1, v=0.09)
        $ 5406 "Set ini_cambro_m289=Encender"
        modbus_set_output_signal("ini_cambro_m289", True)
        $ 5407 "Wait: 2.0"
        sleep(2.0)
        $ 5409 "Wait: 2.0"
        sleep(2.0)
        $ 5410 "Set ini_cambro_m289=Apagar"
        modbus_set_output_signal("ini_cambro_m289", False)
        $ 5411 "Wait: 0.5"
        sleep(0.5)
        $ 5412 "Wait fciclocarr_m292=LO"
        while (modbus_get_signal_status("fciclocarr_m292") == True):
          sync()
        end
        $ 5413 "Wait: 0.5"
        sleep(0.5)
        $ 5415 "MoveL"
        $ 5416 "Precambio_broca" "breakAfter"
        movel(Precambio_broca_p, a=0.1, v=0.09)
        $ 5417 "If eje7≟3"
        if (eje7 == 3):
          $ 5418 "Precam_bro2" "breakAfter"
          movel(Precam_bro2_p, a=1.2, v=0.25)
          $ 5419 "Precam_bro1" "breakAfter"
          movel(Precam_bro1_p, a=1.2, v=0.25)
          $ 5420 "Home3" "breakAfter"
          movel(Home3_p, a=1.2, v=0.25)
        end
        $ 5421 "If eje7≟2"
        if (eje7 == 2):
          $ 5423 "Home2" "breakAfter"
          movel(Home2_p, a=1.2, v=0.25)
        end
        $ 5424 "barrenos_hechos≔0"
        global barrenos_hechos=0
      else:
        $ 5425 "Else" "noBreak"
        $ 5426 "'Codigo de poner broca'"
        # 'Codigo de poner broca'
        $ 5427 "Set ini_cambro_m289=Apagar"
        modbus_set_output_signal("ini_cambro_m289", False)
        $ 5428 "MoveL"
        $ 5429 "Precambio_broca" "breakAfter"
        movel(Precambio_broca_p, a=1.2, v=0.25)
        $ 5430 "Popup: Cambia a las siguientes brocas"
        popup("Cambia a las siguientes brocas", "Advertencia", True, False, blocking=True)
        $ 5431 "Dejar_broca" "breakAfter"
        movel(Dejar_broca_p, a=0.1, v=0.09)
        $ 5432 "Set ini_cambro_m289=Encender"
        modbus_set_output_signal("ini_cambro_m289", True)
        $ 5433 "Wait: 2.0"
        sleep(2.0)
        $ 5435 "Wait: 2.0"
        sleep(2.0)
        $ 5436 "Set ini_cambro_m289=Apagar"
        modbus_set_output_signal("ini_cambro_m289", False)
        $ 5437 "Wait: 0.5"
        sleep(0.5)
        $ 5438 "Wait fciclocarr_m292=LO"
        while (modbus_get_signal_status("fciclocarr_m292") == True):
          sync()
        end
        $ 5439 "Wait: 0.5"
        sleep(0.5)
        $ 5441 "MoveL"
        $ 5442 "Precambio_broca" "breakAfter"
        movel(Precambio_broca_p, a=0.1, v=0.09)
        $ 5443 "If eje7≟3"
        if (eje7 == 3):
          $ 5444 "Precam_bro2" "breakAfter"
          movel(Precam_bro2_p, a=1.2, v=0.25)
          $ 5445 "Precam_bro1" "breakAfter"
          movel(Precam_bro1_p, a=1.2, v=0.25)
          $ 5446 "Home3" "breakAfter"
          movel(Home3_p, a=1.2, v=0.25)
        end
        $ 5447 "If eje7≟2"
        if (eje7 == 2):
          $ 5449 "Home2" "breakAfter"
          movel(Home2_p, a=1.2, v=0.25)
        end
        $ 5450 "barrenos_hechos≔0"
        global barrenos_hechos=0
        $ 5451 "iniciando_prog≔ False "
        global iniciando_prog=  False
        $ 5452 "cambiar_broca≔ False "
        global cambiar_broca=  False
        $ 5453 "Force"
        sleep(0.02)
        zero_ftsensor()
        force_mode(tool_pose(), [0, 0, 1, 0, 0, 0], [0.0, 1.0, 220.0, 0.0, 0.0, 0.0], 2, [0.1, 0.1, 0.15, 0.3490658503988659, 0.3490658503988659, 0.3490658503988659])
        $ 5454 "MoveL" "noBreak"
        $ 5455 "Direction: Base Z-" "noBreak"
        global move_thread_flag_5455=0
        thread move_thread_5455():
          enter_critical
          move_thread_flag_5455 = 1
          local towardsPos=calculate_point_to_move_towards(p[0.0,0.0,0.0,0.0,0.0,0.0], [0.0,0.0,-1.0], 0.024)
          movel(towardsPos, a=1.2, v=0.25)
          move_thread_flag_5455 = 2
          exit_critical
        end
        move_thread_flag_5455 = 0
        move_thread_han_5455 = run move_thread_5455()
        while (True):
          sleep(1.0E-10)
          if (move_thread_flag_5455 > 1):
            join move_thread_han_5455
            $ 5456 "Until (distance)" "noBreak"
            break
          end
          sync()
        end
        end_force_mode()
        stopl(5.0)
      end
    end
  end
  while (True):
    $ 1 "Robot Program"
    $ 2 "Variables"
    $ 3 "bajada_broca≔p[0,0,-0.008,0,0,0]"
    global bajada_broca=p[0,0,-0.008,0,0,0]
    $ 4 "barrenos_menos1≔0"
    global barrenos_menos1=0
    $ 5 "barreno_actual≔0"
    global barreno_actual=0
    $ 6 "posicion≔p[0,0,300,0,0,0]"
    global posicion=p[0,0,300,0,0,0]
    $ 7 "cambiar_broca≔ False "
    global cambiar_broca=  False
    $ 8 "barrenos_hechos≔0"
    global barrenos_hechos=0
    $ 9 "eje7≔0"
    global eje7=0
    $ 10 "Wait: 0.5"
    sleep(0.5)
    $ 11 "Home"
    $ 12 "Wait: 0.3"
    sleep(0.3)
    $ 13 "MoveL"
    $ 14 "Traslacion" "breakAfter"
    movel(Traslacion_p, a=1.2, v=0.25)
    $ 15 "Home2" "breakAfter"
    movel(Home2_p, a=1.2, v=0.25)
    $ 16 "Home3" "breakAfter"
    movel(Home3_p, a=1.2, v=0.25)
    $ 17 "Home4" "breakAfter"
    movel(Home4_p, a=1.2, v=0.25)
    $ 18 "PosicionApagado" "breakAfter"
    movel(PosicionApagado_p, a=1.2, v=0.25)
    $ 19 "Precambio_broca" "breakAfter"
    movel(Precambio_broca_p, a=1.2, v=0.25)
    $ 20 "Home"
    movej([-2.5890958934427104, -1.990702925865989, 2.190075797821148, -0.17834602565650215, -5.748178516127443, -0.01395064457738826], a=1.3962634015954636, v=1.0471975511965976)
    $ 23 "Wait: 0.3"
    sleep(0.3)
    $ 24 "iniciando_prog≔ True "
    global iniciando_prog=  True
    $ 25 "Call Poner_broca"
    Poner_broca()
    $ 26 "Posicion2"
    $ 27 "Inicio"
    $ 28 "eje7≔2"
    global eje7=2
    $ 29 "MoveL"
    $ 30 "Home2" "breakAfter"
    movel(Home2_p, a=1.2, v=0.25)
    $ 31 "SeatTracks"
    $ 32 "Broca_1"
    $ 33 "Linea1"
    $ 34 "Marcar_puntos"
    $ 35 "MoveL"
    $ 36 "Home2" "breakAfter"
    movel(Home2_p, a=0.5, v=0.1)
    $ 37 "Linea1_A" "breakAfter"
    movel(Linea1_A_p, a=0.5, v=0.1)
    $ 38 "Linea1_B" "breakAfter"
    movel(Linea1_B_p, a=0.5, v=0.1)
    $ 39 "Linea1_C" "breakAfter"
    movel(Linea1_C_p, a=0.5, v=0.1)
    $ 40 "Linea1_D" "breakAfter"
    movel(Linea1_D_p, a=0.5, v=0.1)
    $ 41 "Linea1_E" "breakAfter"
    movel(Linea1_E_p, a=0.5, v=0.1)
    $ 42 "Linea1_F" "breakAfter"
    movel(Linea1_F_p, a=0.5, v=0.1)
    $ 43 "AB"
    $ 44 "'desbaste_inicial'"
    # 'desbaste_inicial'
    $ 45 "bajada_broca≔p[0,0,-0.008,0,0,0]"
    global bajada_broca=p[0,0,-0.008,0,0,0]
    $ 46 "barrenos_menos1≔8"
    global barrenos_menos1=8
    $ 47 "barreno_actual≔0"
    global barreno_actual=0
    $ 48 "Loop barreno_actual≤barrenos_menos1"
    while (barreno_actual <= barrenos_menos1):
      $ 49 "Perforacion"
      $ 50 "MoveL"
      $ 51 "internos≔interpolate_pose(Linea1_A, Linea1_B, barreno_actual/barrenos_menos1)"
      global internos= interpolate_pose (Linea1_A_p, Linea1_B_p, barreno_actual/barrenos_menos1)
      $ 52 "internos" "breakAfter"
      movel(internos, a=0.5, v=0.1)
      $ 53 "'desbaste_inicial'"
      # 'desbaste_inicial'
      $ 54 "bajada_broca≔p[0,0,-0.008,0,0,0]"
      global bajada_broca=p[0,0,-0.008,0,0,0]
      $ 55 "bajada≔p[0,0,0.008,0,0,0]"
      global bajada=p[0,0,0.008,0,0,0]
      $ 56 "Direction: Base Z-"
      global move_thread_flag_56=0
      thread move_thread_56():
        enter_critical
        move_thread_flag_56 = 1
        local towardsPos=calculate_point_to_move_towards(p[0.0,0.0,0.0,0.0,0.0,0.0], [0.0,0.0,-1.0], 0.076)
        movel(towardsPos, a=0.015, v=0.015)
        move_thread_flag_56 = 2
        exit_critical
      end
      move_thread_flag_56 = 0
      move_thread_han_56 = run move_thread_56()
      while (True):
        sleep(1.0E-10)
        if (move_thread_flag_56 > 1):
          join move_thread_han_56
          $ 57 "Until (distance)"
          break
        end
        sync()
      end
      $ 58 "Popup: punto contacto alanzdo"
      popup("punto contacto alanzdo", "Mensaje", False, False, blocking=True)
      $ 59 "Direction: Base Z+"
      global move_thread_flag_59=0
      thread move_thread_59():
        enter_critical
        move_thread_flag_59 = 1
        local towardsPos=calculate_point_to_move_towards(p[0.0,0.0,0.0,0.0,0.0,0.0], [0.0,0.0,1.0], 0.002)
        movel(towardsPos, a=0.015, v=0.015)
        move_thread_flag_59 = 2
        exit_critical
      end
      move_thread_flag_59 = 0
      move_thread_han_59 = run move_thread_59()
      while (True):
        sleep(1.0E-10)
        if (move_thread_flag_59 > 1):
          join move_thread_han_59
          $ 60 "Until (distance)"
          break
        end
        sync()
      end
      $ 61 "Wait: 0.3"
      sleep(0.3)
      $ 62 "Set CO[1]=Encender"
      set_configurable_digital_out(1, True)
      $ 63 "Wait: 0.3"
      sleep(0.3)
      $ 64 "Loop 3 times"
      Loop_39 = 0
      while (Loop_39 < 3):
        $ 65 "bajar≔pose_add(get_actual_tcp_pose(), bajada_broca)"
        global bajar= pose_add ( get_actual_tcp_pose (), bajada_broca)
        $ 66 "bajar" "breakAfter"
        movel(bajar, a=0.005, v=0.001)
        $ 67 "subir≔pose_sub(get_actual_tcp_pose(), bajada_broca)"
        global subir= pose_sub ( get_actual_tcp_pose (), bajada_broca)
        $ 68 "subir" "breakAfter"
        movel(subir, a=0.01, v=0.005)
        $ 69 "bajada_broca≔pose_sub(bajada_broca, bajada)"
        global bajada_broca= pose_sub (bajada_broca, bajada)
        Loop_39 = Loop_39 + 1
      end
      $ 70 "Direction: Base Z+"
      global move_thread_flag_70=0
      thread move_thread_70():
        enter_critical
        move_thread_flag_70 = 1
        local towardsPos=calculate_point_to_move_towards(p[0.0,0.0,0.0,0.0,0.0,0.0], [0.0,0.0,1.0], 0.06)
        movel(towardsPos, a=0.035, v=0.03)
        move_thread_flag_70 = 2
        exit_critical
      end
      move_thread_flag_70 = 0
      move_thread_han_70 = run move_thread_70()
      while (True):
        sleep(1.0E-10)
        if (move_thread_flag_70 > 1):
          join move_thread_han_70
          $ 71 "Until (distance)"
          break
        end
        sync()
      end
      $ 72 "Set CO[1]=Apagar"
      set_configurable_digital_out(1, False)
      $ 73 "barreno_actual≔barreno_actual+1"
      global barreno_actual=barreno_actual+1
    end
    $ 76 "CD"
    $ 77 "'desbaste_inicial'"
    # 'desbaste_inicial'
    $ 78 "bajada_broca≔p[0,0,-0.008,0,0,0]"
    global bajada_broca=p[0,0,-0.008,0,0,0]
    $ 79 "barrenos_menos1≔8"
    global barrenos_menos1=8
    $ 80 "barreno_actual≔0"
    global barreno_actual=0
    $ 81 "Loop barreno_actual≤barrenos_menos1"
    while (barreno_actual <= barrenos_menos1):
      $ 82 "Perforacion"
      $ 83 "MoveL"
      $ 84 "internos≔interpolate_pose(Linea1_C, Linea1_D, barreno_actual/barrenos_menos1)"
      global internos= interpolate_pose (Linea1_C_p, Linea1_D_p, barreno_actual/barrenos_menos1)
      $ 85 "internos" "breakAfter"
      movel(internos, a=0.5, v=0.1)
      $ 86 "'desbaste_inicial'"
      # 'desbaste_inicial'
      $ 87 "bajada_broca≔p[0,0,-0.008,0,0,0]"
      global bajada_broca=p[0,0,-0.008,0,0,0]
      $ 88 "bajada≔p[0,0,0.008,0,0,0]"
      global bajada=p[0,0,0.008,0,0,0]
      $ 89 "Direction: Base Z-"
      global move_thread_flag_89=0
      thread move_thread_89():
        enter_critical
        move_thread_flag_89 = 1
        local towardsPos=calculate_point_to_move_towards(p[0.0,0.0,0.0,0.0,0.0,0.0], [0.0,0.0,-1.0], 0.076)
        movel(towardsPos, a=0.015, v=0.015)
        move_thread_flag_89 = 2
        exit_critical
      end
      move_thread_flag_89 = 0
      move_thread_han_89 = run move_thread_89()
      while (True):
        sleep(1.0E-10)
        if (move_thread_flag_89 > 1):
          join move_thread_han_89
          $ 90 "Until (distance)"
          break
        end
        sync()
      end
      $ 91 "Popup: punto contacto alanzdo"
      popup("punto contacto alanzdo", "Mensaje", False, False, blocking=True)
      $ 92 "Direction: Base Z+"
      global move_thread_flag_92=0
      thread move_thread_92():
        enter_critical
        move_thread_flag_92 = 1
        local towardsPos=calculate_point_to_move_towards(p[0.0,0.0,0.0,0.0,0.0,0.0], [0.0,0.0,1.0], 0.002)
        movel(towardsPos, a=0.005, v=0.003)
        move_thread_flag_92 = 2
        exit_critical
      end
      move_thread_flag_92 = 0
      move_thread_han_92 = run move_thread_92()
      while (True):
        sleep(1.0E-10)
        if (move_thread_flag_92 > 1):
          join move_thread_han_92
          $ 93 "Until (distance)"
          break
        end
        sync()
      end
      $ 94 "Wait: 0.3"
      sleep(0.3)
      $ 95 "Set CO[1]=Encender"
      set_configurable_digital_out(1, True)
      $ 96 "Wait: 0.3"
      sleep(0.3)
      $ 97 "Loop 3 times"
      Loop_56 = 0
      while (Loop_56 < 3):
        $ 98 "bajar≔pose_add(get_actual_tcp_pose(), bajada_broca)"
        global bajar= pose_add ( get_actual_tcp_pose (), bajada_broca)
        $ 99 "bajar" "breakAfter"
        movel(bajar, a=0.005, v=0.001)
        $ 100 "subir≔pose_sub(get_actual_tcp_pose(), bajada_broca)"
        global subir= pose_sub ( get_actual_tcp_pose (), bajada_broca)
        $ 101 "subir" "breakAfter"
        movel(subir, a=0.01, v=0.005)
        $ 102 "bajada_broca≔pose_sub(bajada_broca, bajada)"
        global bajada_broca= pose_sub (bajada_broca, bajada)
        Loop_56 = Loop_56 + 1
      end
      $ 103 "Direction: Base Z+"
      global move_thread_flag_103=0
      thread move_thread_103():
        enter_critical
        move_thread_flag_103 = 1
        local towardsPos=calculate_point_to_move_towards(p[0.0,0.0,0.0,0.0,0.0,0.0], [0.0,0.0,1.0], 0.06)
        movel(towardsPos, a=0.035, v=0.03)
        move_thread_flag_103 = 2
        exit_critical
      end
      move_thread_flag_103 = 0
      move_thread_han_103 = run move_thread_103()
      while (True):
        sleep(1.0E-10)
        if (move_thread_flag_103 > 1):
          join move_thread_han_103
          $ 104 "Until (distance)"
          break
        end
        sync()
      end
      $ 105 "Set CO[1]=Apagar"
      set_configurable_digital_out(1, False)
      $ 106 "barreno_actual≔barreno_actual+1"
      global barreno_actual=barreno_actual+1
    end
    $ 109 "EF"
    $ 110 "'desbaste_inicial'"
    # 'desbaste_inicial'
    $ 111 "bajada_broca≔p[0,0,-0.008,0,0,0]"
    global bajada_broca=p[0,0,-0.008,0,0,0]
    $ 112 "barrenos_menos1≔8"
    global barrenos_menos1=8
    $ 113 "barreno_actual≔0"
    global barreno_actual=0
    $ 114 "Loop barreno_actual≤barrenos_menos1"
    while (barreno_actual <= barrenos_menos1):
      $ 115 "Perforacion"
      $ 116 "MoveL"
      $ 117 "internos≔interpolate_pose(Linea1_E, Linea1_F, barreno_actual/barrenos_menos1)"
      global internos= interpolate_pose (Linea1_E_p, Linea1_F_p, barreno_actual/barrenos_menos1)
      $ 118 "internos" "breakAfter"
      movel(internos, a=0.5, v=0.1)
      $ 119 "'desbaste_inicial'"
      # 'desbaste_inicial'
      $ 120 "bajada_broca≔p[0,0,-0.008,0,0,0]"
      global bajada_broca=p[0,0,-0.008,0,0,0]
      $ 121 "bajada≔p[0,0,0.008,0,0,0]"
      global bajada=p[0,0,0.008,0,0,0]
      $ 122 "Direction: Base Z-"
      global move_thread_flag_122=0
      thread move_thread_122():
        enter_critical
        move_thread_flag_122 = 1
        local towardsPos=calculate_point_to_move_towards(p[0.0,0.0,0.0,0.0,0.0,0.0], [0.0,0.0,-1.0], 0.076)
        movel(towardsPos, a=0.015, v=0.015)
        move_thread_flag_122 = 2
        exit_critical
      end
      move_thread_flag_122 = 0
      move_thread_han_122 = run move_thread_122()
      while (True):
        sleep(1.0E-10)
        if (move_thread_flag_122 > 1):
          join move_thread_han_122
          $ 123 "Until (distance)"
          break
        end
        sync()
      end
      $ 124 "Popup: punto contacto alanzdo"
      popup("punto contacto alanzdo", "Mensaje", False, False, blocking=True)
      $ 125 "Direction: Base Z+"
      global move_thread_flag_125=0
      thread move_thread_125():
        enter_critical
        move_thread_flag_125 = 1
        local towardsPos=calculate_point_to_move_towards(p[0.0,0.0,0.0,0.0,0.0,0.0], [0.0,0.0,1.0], 0.002)
        movel(towardsPos, a=0.005, v=0.003)
        move_thread_flag_125 = 2
        exit_critical
      end
      move_thread_flag_125 = 0
      move_thread_han_125 = run move_thread_125()
      while (True):
        sleep(1.0E-10)
        if (move_thread_flag_125 > 1):
          join move_thread_han_125
          $ 126 "Until (distance)"
          break
        end
        sync()
      end
      $ 127 "Wait: 0.3"
      sleep(0.3)
      $ 128 "Set CO[1]=Encender"
      set_configurable_digital_out(1, True)
      $ 129 "Wait: 0.3"
      sleep(0.3)
      $ 130 "Loop 3 times"
      Loop_61 = 0
      while (Loop_61 < 3):
        $ 131 "bajar≔pose_add(get_actual_tcp_pose(), bajada_broca)"
        global bajar= pose_add ( get_actual_tcp_pose (), bajada_broca)
        $ 132 "bajar" "breakAfter"
        movel(bajar, a=0.005, v=0.001)
        $ 133 "subir≔pose_sub(get_actual_tcp_pose(), bajada_broca)"
        global subir= pose_sub ( get_actual_tcp_pose (), bajada_broca)
        $ 134 "subir" "breakAfter"
        movel(subir, a=0.01, v=0.005)
        $ 135 "bajada_broca≔pose_sub(bajada_broca, bajada)"
        global bajada_broca= pose_sub (bajada_broca, bajada)
        Loop_61 = Loop_61 + 1
      end
      $ 136 "Direction: Base Z+"
      global move_thread_flag_136=0
      thread move_thread_136():
        enter_critical
        move_thread_flag_136 = 1
        local towardsPos=calculate_point_to_move_towards(p[0.0,0.0,0.0,0.0,0.0,0.0], [0.0,0.0,1.0], 0.06)
        movel(towardsPos, a=0.035, v=0.03)
        move_thread_flag_136 = 2
        exit_critical
      end
      move_thread_flag_136 = 0
      move_thread_han_136 = run move_thread_136()
      while (True):
        sleep(1.0E-10)
        if (move_thread_flag_136 > 1):
          join move_thread_han_136
          $ 137 "Until (distance)"
          break
        end
        sync()
      end
      $ 138 "Set CO[1]=Apagar"
      set_configurable_digital_out(1, False)
      $ 139 "barreno_actual≔barreno_actual+1"
      global barreno_actual=barreno_actual+1
    end
    $ 142 "Popup: Linea1 con chica Terminada!"
    popup("Linea1 con chica Terminada!", "Mensaje", False, False, blocking=True)
    $ 143 "Linea2"
    $ 144 "Marcar_puntos"
    $ 145 "MoveL"
    $ 146 "Home2" "breakAfter"
    movel(Home2_p, a=0.5, v=0.1)
    $ 147 "Linea2_A" "breakAfter"
    movel(Linea2_A_p, a=0.5, v=0.1)
    $ 148 "Linea2_B" "breakAfter"
    movel(Linea2_B_p, a=0.5, v=0.1)
    $ 149 "Linea2_C" "breakAfter"
    movel(Linea2_C_p, a=0.5, v=0.1)
    $ 150 "Linea2_D" "breakAfter"
    movel(Linea2_D_p, a=0.5, v=0.1)
    $ 151 "Linea2_E" "breakAfter"
    movel(Linea2_E_p, a=0.5, v=0.1)
    $ 152 "Linea2_F" "breakAfter"
    movel(Linea2_F_p, a=0.5, v=0.1)
    $ 153 "AB"
    $ 154 "'desbaste_inicial'"
    # 'desbaste_inicial'
    $ 155 "bajada_broca≔p[0,0,-0.008,0,0,0]"
    global bajada_broca=p[0,0,-0.008,0,0,0]
    $ 156 "barrenos_menos1≔8"
    global barrenos_menos1=8
    $ 157 "barreno_actual≔0"
    global barreno_actual=0
    $ 158 "Loop barreno_actual≤barrenos_menos1"
    while (barreno_actual <= barrenos_menos1):
      $ 159 "Perforacion"
      $ 160 "MoveL"
      $ 161 "internos≔interpolate_pose(Linea2_A, Linea2_B, barreno_actual/barrenos_menos1)"
      global internos= interpolate_pose (Linea2_A_p, Linea2_B_p, barreno_actual/barrenos_menos1)
      $ 162 "internos" "breakAfter"
      movel(internos, a=0.5, v=0.1)
      $ 163 "'desbaste_inicial'"
      # 'desbaste_inicial'
      $ 164 "bajada_broca≔p[0,0,-0.008,0,0,0]"
      global bajada_broca=p[0,0,-0.008,0,0,0]
      $ 165 "bajada≔p[0,0,0.008,0,0,0]"
      global bajada=p[0,0,0.008,0,0,0]
      $ 166 "Direction: Base Z-"
      global move_thread_flag_166=0
      thread move_thread_166():
        enter_critical
        move_thread_flag_166 = 1
        local towardsPos=calculate_point_to_move_towards(p[0.0,0.0,0.0,0.0,0.0,0.0], [0.0,0.0,-1.0], 0.076)
        movel(towardsPos, a=0.015, v=0.015)
        move_thread_flag_166 = 2
        exit_critical
      end
      move_thread_flag_166 = 0
      move_thread_han_166 = run move_thread_166()
      while (True):
        sleep(1.0E-10)
        if (move_thread_flag_166 > 1):
          join move_thread_han_166
          $ 167 "Until (distance)"
          break
        end
        sync()
      end
      $ 168 "Popup: punto contacto alanzdo"
      popup("punto contacto alanzdo", "Mensaje", False, False, blocking=True)
      $ 169 "Direction: Base Z+"
      global move_thread_flag_169=0
      thread move_thread_169():
        enter_critical
        move_thread_flag_169 = 1
        local towardsPos=calculate_point_to_move_towards(p[0.0,0.0,0.0,0.0,0.0,0.0], [0.0,0.0,1.0], 0.002)
        movel(towardsPos, a=0.005, v=0.003)
        move_thread_flag_169 = 2
        exit_critical
      end
      move_thread_flag_169 = 0
      move_thread_han_169 = run move_thread_169()
      while (True):
        sleep(1.0E-10)
        if (move_thread_flag_169 > 1):
          join move_thread_han_169
          $ 170 "Until (distance)"
          break
        end
        sync()
      end
      $ 171 "Wait: 0.3"
      sleep(0.3)
      $ 172 "Set CO[1]=Encender"
      set_configurable_digital_out(1, True)
      $ 173 "Wait: 0.3"
      sleep(0.3)
      $ 174 "Loop 3 times"
      Loop_63 = 0
      while (Loop_63 < 3):
        $ 175 "bajar≔pose_add(get_actual_tcp_pose(), bajada_broca)"
        global bajar= pose_add ( get_actual_tcp_pose (), bajada_broca)
        $ 176 "bajar" "breakAfter"
        movel(bajar, a=0.005, v=0.001)
        $ 177 "subir≔pose_sub(get_actual_tcp_pose(), bajada_broca)"
        global subir= pose_sub ( get_actual_tcp_pose (), bajada_broca)
        $ 178 "subir" "breakAfter"
        movel(subir, a=0.01, v=0.005)
        $ 179 "bajada_broca≔pose_sub(bajada_broca, bajada)"
        global bajada_broca= pose_sub (bajada_broca, bajada)
        Loop_63 = Loop_63 + 1
      end
      $ 180 "Direction: Base Z+"
      global move_thread_flag_180=0
      thread move_thread_180():
        enter_critical
        move_thread_flag_180 = 1
        local towardsPos=calculate_point_to_move_towards(p[0.0,0.0,0.0,0.0,0.0,0.0], [0.0,0.0,1.0], 0.06)
        movel(towardsPos, a=0.035, v=0.03)
        move_thread_flag_180 = 2
        exit_critical
      end
      move_thread_flag_180 = 0
      move_thread_han_180 = run move_thread_180()
      while (True):
        sleep(1.0E-10)
        if (move_thread_flag_180 > 1):
          join move_thread_han_180
          $ 181 "Until (distance)"
          break
        end
        sync()
      end
      $ 182 "Set CO[1]=Apagar"
      set_configurable_digital_out(1, False)
      $ 183 "barreno_actual≔barreno_actual+1"
      global barreno_actual=barreno_actual+1
    end
    $ 186 "CD"
    $ 187 "'desbaste_inicial'"
    # 'desbaste_inicial'
    $ 188 "bajada_broca≔p[0,0,-0.008,0,0,0]"
    global bajada_broca=p[0,0,-0.008,0,0,0]
    $ 189 "barrenos_menos1≔8"
    global barrenos_menos1=8
    $ 190 "barreno_actual≔0"
    global barreno_actual=0
    $ 191 "Loop barreno_actual≤barrenos_menos1"
    while (barreno_actual <= barrenos_menos1):
      $ 192 "Perforacion"
      $ 193 "MoveL"
      $ 194 "internos≔interpolate_pose(Linea2_C, Linea2_D, barreno_actual/barrenos_menos1)"
      global internos= interpolate_pose (Linea2_C_p, Linea2_D_p, barreno_actual/barrenos_menos1)
      $ 195 "internos" "breakAfter"
      movel(internos, a=0.5, v=0.1)
      $ 196 "'desbaste_inicial'"
      # 'desbaste_inicial'
      $ 197 "bajada_broca≔p[0,0,-0.008,0,0,0]"
      global bajada_broca=p[0,0,-0.008,0,0,0]
      $ 198 "bajada≔p[0,0,0.008,0,0,0]"
      global bajada=p[0,0,0.008,0,0,0]
      $ 199 "Direction: Base Z-"
      global move_thread_flag_199=0
      thread move_thread_199():
        enter_critical
        move_thread_flag_199 = 1
        local towardsPos=calculate_point_to_move_towards(p[0.0,0.0,0.0,0.0,0.0,0.0], [0.0,0.0,-1.0], 0.076)
        movel(towardsPos, a=0.015, v=0.015)
        move_thread_flag_199 = 2
        exit_critical
      end
      move_thread_flag_199 = 0
      move_thread_han_199 = run move_thread_199()
      while (True):
        sleep(1.0E-10)
        if (move_thread_flag_199 > 1):
          join move_thread_han_199
          $ 200 "Until (distance)"
          break
        end
        sync()
      end
      $ 201 "Popup: punto contacto alanzdo"
      popup("punto contacto alanzdo", "Mensaje", False, False, blocking=True)
      $ 202 "Direction: Base Z+"
      global move_thread_flag_202=0
      thread move_thread_202():
        enter_critical
        move_thread_flag_202 = 1
        local towardsPos=calculate_point_to_move_towards(p[0.0,0.0,0.0,0.0,0.0,0.0], [0.0,0.0,1.0], 0.002)
        movel(towardsPos, a=0.005, v=0.003)
        move_thread_flag_202 = 2
        exit_critical
      end
      move_thread_flag_202 = 0
      move_thread_han_202 = run move_thread_202()
      while (True):
        sleep(1.0E-10)
        if (move_thread_flag_202 > 1):
          join move_thread_han_202
          $ 203 "Until (distance)"
          break
        end
        sync()
      end
      $ 204 "Wait: 0.3"
      sleep(0.3)
      $ 205 "Set CO[1]=Encender"
      set_configurable_digital_out(1, True)
      $ 206 "Wait: 0.3"
      sleep(0.3)
      $ 207 "Loop 3 times"
      Loop_65 = 0
      while (Loop_65 < 3):
        $ 208 "bajar≔pose_add(get_actual_tcp_pose(), bajada_broca)"
        global bajar= pose_add ( get_actual_tcp_pose (), bajada_broca)
        $ 209 "bajar" "breakAfter"
        movel(bajar, a=0.005, v=0.001)
        $ 210 "subir≔pose_sub(get_actual_tcp_pose(), bajada_broca)"
        global subir= pose_sub ( get_actual_tcp_pose (), bajada_broca)
        $ 211 "subir" "breakAfter"
        movel(subir, a=0.01, v=0.005)
        $ 212 "bajada_broca≔pose_sub(bajada_broca, bajada)"
        global bajada_broca= pose_sub (bajada_broca, bajada)
        Loop_65 = Loop_65 + 1
      end
      $ 213 "Direction: Base Z+"
      global move_thread_flag_213=0
      thread move_thread_213():
        enter_critical
        move_thread_flag_213 = 1
        local towardsPos=calculate_point_to_move_towards(p[0.0,0.0,0.0,0.0,0.0,0.0], [0.0,0.0,1.0], 0.06)
        movel(towardsPos, a=0.035, v=0.03)
        move_thread_flag_213 = 2
        exit_critical
      end
      move_thread_flag_213 = 0
      move_thread_han_213 = run move_thread_213()
      while (True):
        sleep(1.0E-10)
        if (move_thread_flag_213 > 1):
          join move_thread_han_213
          $ 214 "Until (distance)"
          break
        end
        sync()
      end
      $ 215 "Set CO[1]=Apagar"
      set_configurable_digital_out(1, False)
      $ 216 "barreno_actual≔barreno_actual+1"
      global barreno_actual=barreno_actual+1
    end
    $ 219 "EF"
    $ 220 "'desbaste_inicial'"
    # 'desbaste_inicial'
    $ 221 "bajada_broca≔p[0,0,-0.008,0,0,0]"
    global bajada_broca=p[0,0,-0.008,0,0,0]
    $ 222 "barrenos_menos1≔8"
    global barrenos_menos1=8
    $ 223 "barreno_actual≔0"
    global barreno_actual=0
    $ 224 "Loop barreno_actual≤barrenos_menos1"
    while (barreno_actual <= barrenos_menos1):
      $ 225 "Perforacion"
      $ 226 "MoveL"
      $ 227 "internos≔interpolate_pose(Linea2_E, Linea2_F, barreno_actual/barrenos_menos1)"
      global internos= interpolate_pose (Linea2_E_p, Linea2_F_p, barreno_actual/barrenos_menos1)
      $ 228 "internos" "breakAfter"
      movel(internos, a=0.5, v=0.1)
      $ 229 "'desbaste_inicial'"
      # 'desbaste_inicial'
      $ 230 "bajada_broca≔p[0,0,-0.008,0,0,0]"
      global bajada_broca=p[0,0,-0.008,0,0,0]
      $ 231 "bajada≔p[0,0,0.008,0,0,0]"
      global bajada=p[0,0,0.008,0,0,0]
      $ 232 "Direction: Base Z-"
      global move_thread_flag_232=0
      thread move_thread_232():
        enter_critical
        move_thread_flag_232 = 1
        local towardsPos=calculate_point_to_move_towards(p[0.0,0.0,0.0,0.0,0.0,0.0], [0.0,0.0,-1.0], 0.076)
        movel(towardsPos, a=0.015, v=0.015)
        move_thread_flag_232 = 2
        exit_critical
      end
      move_thread_flag_232 = 0
      move_thread_han_232 = run move_thread_232()
      while (True):
        sleep(1.0E-10)
        if (move_thread_flag_232 > 1):
          join move_thread_han_232
          $ 233 "Until (distance)"
          break
        end
        sync()
      end
      $ 234 "Popup: punto contacto alanzdo"
      popup("punto contacto alanzdo", "Mensaje", False, False, blocking=True)
      $ 235 "Direction: Base Z+"
      global move_thread_flag_235=0
      thread move_thread_235():
        enter_critical
        move_thread_flag_235 = 1
        local towardsPos=calculate_point_to_move_towards(p[0.0,0.0,0.0,0.0,0.0,0.0], [0.0,0.0,1.0], 0.002)
        movel(towardsPos, a=0.005, v=0.003)
        move_thread_flag_235 = 2
        exit_critical
      end
      move_thread_flag_235 = 0
      move_thread_han_235 = run move_thread_235()
      while (True):
        sleep(1.0E-10)
        if (move_thread_flag_235 > 1):
          join move_thread_han_235
          $ 236 "Until (distance)"
          break
        end
        sync()
      end
      $ 237 "Wait: 0.3"
      sleep(0.3)
      $ 238 "Set CO[1]=Encender"
      set_configurable_digital_out(1, True)
      $ 239 "Wait: 0.3"
      sleep(0.3)
      $ 240 "Loop 3 times"
      Loop_67 = 0
      while (Loop_67 < 3):
        $ 241 "bajar≔pose_add(get_actual_tcp_pose(), bajada_broca)"
        global bajar= pose_add ( get_actual_tcp_pose (), bajada_broca)
        $ 242 "bajar" "breakAfter"
        movel(bajar, a=0.005, v=0.001)
        $ 243 "subir≔pose_sub(get_actual_tcp_pose(), bajada_broca)"
        global subir= pose_sub ( get_actual_tcp_pose (), bajada_broca)
        $ 244 "subir" "breakAfter"
        movel(subir, a=0.01, v=0.005)
        $ 245 "bajada_broca≔pose_sub(bajada_broca, bajada)"
        global bajada_broca= pose_sub (bajada_broca, bajada)
        Loop_67 = Loop_67 + 1
      end
      $ 246 "Direction: Base Z+"
      global move_thread_flag_246=0
      thread move_thread_246():
        enter_critical
        move_thread_flag_246 = 1
        local towardsPos=calculate_point_to_move_towards(p[0.0,0.0,0.0,0.0,0.0,0.0], [0.0,0.0,1.0], 0.06)
        movel(towardsPos, a=0.035, v=0.03)
        move_thread_flag_246 = 2
        exit_critical
      end
      move_thread_flag_246 = 0
      move_thread_han_246 = run move_thread_246()
      while (True):
        sleep(1.0E-10)
        if (move_thread_flag_246 > 1):
          join move_thread_han_246
          $ 247 "Until (distance)"
          break
        end
        sync()
      end
      $ 248 "Set CO[1]=Apagar"
      set_configurable_digital_out(1, False)
      $ 249 "barreno_actual≔barreno_actual+1"
      global barreno_actual=barreno_actual+1
      $ 250 "If barreno_actual≥barrenos_menos1"
      if (barreno_actual >= barrenos_menos1):
        $ 251 "cambiar_broca≔ True "
        global cambiar_broca=  True
      end
    end
    $ 254 "Popup: Linea2 con chica Terminada!"
    popup("Linea2 con chica Terminada!", "Mensaje", False, False, blocking=True)
    $ 255 "Broca_2"
    $ 256 "Linea1"
    $ 257 "Marcar_puntos"
    $ 258 "MoveL"
    $ 259 "Home2" "breakAfter"
    movel(Home2_p, a=0.5, v=0.1)
    $ 260 "Linea1_A" "breakAfter"
    movel(Linea1_A_p, a=0.5, v=0.1)
    $ 261 "Linea1_B" "breakAfter"
    movel(Linea1_B_p, a=0.5, v=0.1)
    $ 262 "Linea1_C" "breakAfter"
    movel(Linea1_C_p, a=0.5, v=0.1)
    $ 263 "Linea1_D" "breakAfter"
    movel(Linea1_D_p, a=0.5, v=0.1)
    $ 264 "Linea1_E" "breakAfter"
    movel(Linea1_E_p, a=0.5, v=0.1)
    $ 265 "Linea1_F" "breakAfter"
    movel(Linea1_F_p, a=0.5, v=0.1)
    $ 266 "AB"
    $ 267 "'desbaste_inicial'"
    # 'desbaste_inicial'
    $ 268 "bajada_broca≔p[0,0,-0.012,0,0,0]"
    global bajada_broca=p[0,0,-0.012,0,0,0]
    $ 269 "barrenos_menos1≔8"
    global barrenos_menos1=8
    $ 270 "barreno_actual≔0"
    global barreno_actual=0
    $ 271 "Loop barreno_actual≤barrenos_menos1"
    while (barreno_actual <= barrenos_menos1):
      $ 272 "Perforacion"
      $ 273 "MoveL"
      $ 274 "internos≔interpolate_pose(Linea1_A, Linea1_B, barreno_actual/barrenos_menos1)"
      global internos= interpolate_pose (Linea1_A_p, Linea1_B_p, barreno_actual/barrenos_menos1)
      $ 275 "internos" "breakAfter"
      movel(internos, a=0.5, v=0.1)
      $ 276 "'desbaste_inicial'"
      # 'desbaste_inicial'
      $ 277 "bajada_broca≔p[0,0,-0.012,0,0,0]"
      global bajada_broca=p[0,0,-0.012,0,0,0]
      $ 278 "bajada≔p[0,0,0.012,0,0,0]"
      global bajada=p[0,0,0.012,0,0,0]
      $ 279 "Direction: Base Z-"
      global move_thread_flag_279=0
      thread move_thread_279():
        enter_critical
        move_thread_flag_279 = 1
        local towardsPos=calculate_point_to_move_towards(p[0.0,0.0,0.0,0.0,0.0,0.0], [0.0,0.0,-1.0], 0.076)
        movel(towardsPos, a=0.015, v=0.015)
        move_thread_flag_279 = 2
        exit_critical
      end
      move_thread_flag_279 = 0
      move_thread_han_279 = run move_thread_279()
      while (True):
        sleep(1.0E-10)
        if (move_thread_flag_279 > 1):
          join move_thread_han_279
          $ 280 "Until (distance)"
          break
        end
        sync()
      end
      $ 281 "Popup: punto contacto alanzdo"
      popup("punto contacto alanzdo", "Mensaje", False, False, blocking=True)
      $ 282 "Direction: Base Z+"
      global move_thread_flag_282=0
      thread move_thread_282():
        enter_critical
        move_thread_flag_282 = 1
        local towardsPos=calculate_point_to_move_towards(p[0.0,0.0,0.0,0.0,0.0,0.0], [0.0,0.0,1.0], 0.002)
        movel(towardsPos, a=0.005, v=0.003)
        move_thread_flag_282 = 2
        exit_critical
      end
      move_thread_flag_282 = 0
      move_thread_han_282 = run move_thread_282()
      while (True):
        sleep(1.0E-10)
        if (move_thread_flag_282 > 1):
          join move_thread_han_282
          $ 283 "Until (distance)"
          break
        end
        sync()
      end
      $ 284 "Wait: 0.3"
      sleep(0.3)
      $ 285 "Set CO[1]=Encender"
      set_configurable_digital_out(1, True)
      $ 286 "Wait: 0.3"
      sleep(0.3)
      $ 287 "Loop 2 times"
      Loop_69 = 0
      while (Loop_69 < 2):
        $ 288 "bajar≔pose_add(get_actual_tcp_pose(), bajada_broca)"
        global bajar= pose_add ( get_actual_tcp_pose (), bajada_broca)
        $ 289 "bajar" "breakAfter"
        movel(bajar, a=0.005, v=0.001)
        $ 290 "subir≔pose_sub(get_actual_tcp_pose(), bajada_broca)"
        global subir= pose_sub ( get_actual_tcp_pose (), bajada_broca)
        $ 291 "subir" "breakAfter"
        movel(subir, a=0.01, v=0.005)
        $ 292 "bajada_broca≔pose_sub(bajada_broca, bajada)"
        global bajada_broca= pose_sub (bajada_broca, bajada)
        Loop_69 = Loop_69 + 1
      end
      $ 293 "Direction: Base Z+"
      global move_thread_flag_293=0
      thread move_thread_293():
        enter_critical
        move_thread_flag_293 = 1
        local towardsPos=calculate_point_to_move_towards(p[0.0,0.0,0.0,0.0,0.0,0.0], [0.0,0.0,1.0], 0.06)
        movel(towardsPos, a=0.035, v=0.03)
        move_thread_flag_293 = 2
        exit_critical
      end
      move_thread_flag_293 = 0
      move_thread_han_293 = run move_thread_293()
      while (True):
        sleep(1.0E-10)
        if (move_thread_flag_293 > 1):
          join move_thread_han_293
          $ 294 "Until (distance)"
          break
        end
        sync()
      end
      $ 295 "Set CO[1]=Apagar"
      set_configurable_digital_out(1, False)
      $ 296 "barreno_actual≔barreno_actual+1"
      global barreno_actual=barreno_actual+1
      $ 297 "Call Quitar_broca"
      Quitar_broca()
      $ 298 "Call Poner_broca"
      Poner_broca()
    end
    $ 299 "CD"
    $ 300 "'desbaste_inicial'"
    # 'desbaste_inicial'
    $ 301 "bajada_broca≔p[0,0,-0.012,0,0,0]"
    global bajada_broca=p[0,0,-0.012,0,0,0]
    $ 302 "barrenos_menos1≔8"
    global barrenos_menos1=8
    $ 303 "barreno_actual≔0"
    global barreno_actual=0
    $ 304 "Loop barreno_actual≤barrenos_menos1"
    while (barreno_actual <= barrenos_menos1):
      $ 305 "Perforacion"
      $ 306 "MoveL"
      $ 307 "internos≔interpolate_pose(Linea1_C, Linea1_D, barreno_actual/barrenos_menos1)"
      global internos= interpolate_pose (Linea1_C_p, Linea1_D_p, barreno_actual/barrenos_menos1)
      $ 308 "internos" "breakAfter"
      movel(internos, a=0.5, v=0.1)
      $ 309 "'desbaste_inicial'"
      # 'desbaste_inicial'
      $ 310 "bajada_broca≔p[0,0,-0.012,0,0,0]"
      global bajada_broca=p[0,0,-0.012,0,0,0]
      $ 311 "bajada≔p[0,0,0.012,0,0,0]"
      global bajada=p[0,0,0.012,0,0,0]
      $ 312 "Direction: Base Z-"
      global move_thread_flag_312=0
      thread move_thread_312():
        enter_critical
        move_thread_flag_312 = 1
        local towardsPos=calculate_point_to_move_towards(p[0.0,0.0,0.0,0.0,0.0,0.0], [0.0,0.0,-1.0], 0.076)
        movel(towardsPos, a=0.015, v=0.015)
        move_thread_flag_312 = 2
        exit_critical
      end
      move_thread_flag_312 = 0
      move_thread_han_312 = run move_thread_312()
      while (True):
        sleep(1.0E-10)
        if (move_thread_flag_312 > 1):
          join move_thread_han_312
          $ 313 "Until (distance)"
          break
        end
        sync()
      end
      $ 314 "Popup: punto contacto alanzdo"
      popup("punto contacto alanzdo", "Mensaje", False, False, blocking=True)
      $ 315 "Direction: Base Z+"
      global move_thread_flag_315=0
      thread move_thread_315():
        enter_critical
        move_thread_flag_315 = 1
        local towardsPos=calculate_point_to_move_towards(p[0.0,0.0,0.0,0.0,0.0,0.0], [0.0,0.0,1.0], 0.002)
        movel(towardsPos, a=0.005, v=0.003)
        move_thread_flag_315 = 2
        exit_critical
      end
      move_thread_flag_315 = 0
      move_thread_han_315 = run move_thread_315()
      while (True):
        sleep(1.0E-10)
        if (move_thread_flag_315 > 1):
          join move_thread_han_315
          $ 316 "Until (distance)"
          break
        end
        sync()
      end
      $ 317 "Wait: 0.3"
      sleep(0.3)
      $ 318 "Set CO[1]=Encender"
      set_configurable_digital_out(1, True)
      $ 319 "Wait: 0.3"
      sleep(0.3)
      $ 320 "Loop 2 times"
      Loop_71 = 0
      while (Loop_71 < 2):
        $ 321 "bajar≔pose_add(get_actual_tcp_pose(), bajada_broca)"
        global bajar= pose_add ( get_actual_tcp_pose (), bajada_broca)
        $ 322 "bajar" "breakAfter"
        movel(bajar, a=0.005, v=0.001)
        $ 323 "subir≔pose_sub(get_actual_tcp_pose(), bajada_broca)"
        global subir= pose_sub ( get_actual_tcp_pose (), bajada_broca)
        $ 324 "subir" "breakAfter"
        movel(subir, a=0.01, v=0.005)
        $ 325 "bajada_broca≔pose_sub(bajada_broca, bajada)"
        global bajada_broca= pose_sub (bajada_broca, bajada)
        Loop_71 = Loop_71 + 1
      end
      $ 326 "Direction: Base Z+"
      global move_thread_flag_326=0
      thread move_thread_326():
        enter_critical
        move_thread_flag_326 = 1
        local towardsPos=calculate_point_to_move_towards(p[0.0,0.0,0.0,0.0,0.0,0.0], [0.0,0.0,1.0], 0.06)
        movel(towardsPos, a=0.035, v=0.03)
        move_thread_flag_326 = 2
        exit_critical
      end
      move_thread_flag_326 = 0
      move_thread_han_326 = run move_thread_326()
      while (True):
        sleep(1.0E-10)
        if (move_thread_flag_326 > 1):
          join move_thread_han_326
          $ 327 "Until (distance)"
          break
        end
        sync()
      end
      $ 328 "Set CO[1]=Apagar"
      set_configurable_digital_out(1, False)
      $ 329 "barreno_actual≔barreno_actual+1"
      global barreno_actual=barreno_actual+1
      $ 330 "Call Quitar_broca"
      Quitar_broca()
      $ 331 "Call Poner_broca"
      Poner_broca()
    end
    $ 332 "EF"
    $ 333 "'desbaste_inicial'"
    # 'desbaste_inicial'
    $ 334 "bajada_broca≔p[0,0,-0.012,0,0,0]"
    global bajada_broca=p[0,0,-0.012,0,0,0]
    $ 335 "barrenos_menos1≔8"
    global barrenos_menos1=8
    $ 336 "barreno_actual≔0"
    global barreno_actual=0
    $ 337 "Loop barreno_actual≤barrenos_menos1"
    while (barreno_actual <= barrenos_menos1):
      $ 338 "Perforacion"
      $ 339 "MoveL"
      $ 340 "internos≔interpolate_pose(Linea1_E, Linea1_F, barreno_actual/barrenos_menos1)"
      global internos= interpolate_pose (Linea1_E_p, Linea1_F_p, barreno_actual/barrenos_menos1)
      $ 341 "internos" "breakAfter"
      movel(internos, a=0.5, v=0.1)
      $ 342 "'desbaste_inicial'"
      # 'desbaste_inicial'
      $ 343 "bajada_broca≔p[0,0,-0.012,0,0,0]"
      global bajada_broca=p[0,0,-0.012,0,0,0]
      $ 344 "bajada≔p[0,0,0.012,0,0,0]"
      global bajada=p[0,0,0.012,0,0,0]
      $ 345 "Direction: Base Z-"
      global move_thread_flag_345=0
      thread move_thread_345():
        enter_critical
        move_thread_flag_345 = 1
        local towardsPos=calculate_point_to_move_towards(p[0.0,0.0,0.0,0.0,0.0,0.0], [0.0,0.0,-1.0], 0.076)
        movel(towardsPos, a=0.015, v=0.015)
        move_thread_flag_345 = 2
        exit_critical
      end
      move_thread_flag_345 = 0
      move_thread_han_345 = run move_thread_345()
      while (True):
        sleep(1.0E-10)
        if (move_thread_flag_345 > 1):
          join move_thread_han_345
          $ 346 "Until (distance)"
          break
        end
        sync()
      end
      $ 347 "Popup: punto contacto alanzdo"
      popup("punto contacto alanzdo", "Mensaje", False, False, blocking=True)
      $ 348 "Direction: Base Z+"
      global move_thread_flag_348=0
      thread move_thread_348():
        enter_critical
        move_thread_flag_348 = 1
        local towardsPos=calculate_point_to_move_towards(p[0.0,0.0,0.0,0.0,0.0,0.0], [0.0,0.0,1.0], 0.002)
        movel(towardsPos, a=0.005, v=0.003)
        move_thread_flag_348 = 2
        exit_critical
      end
      move_thread_flag_348 = 0
      move_thread_han_348 = run move_thread_348()
      while (True):
        sleep(1.0E-10)
        if (move_thread_flag_348 > 1):
          join move_thread_han_348
          $ 349 "Until (distance)"
          break
        end
        sync()
      end
      $ 350 "Wait: 0.3"
      sleep(0.3)
      $ 351 "Set CO[1]=Encender"
      set_configurable_digital_out(1, True)
      $ 352 "Wait: 0.3"
      sleep(0.3)
      $ 353 "Loop 2 times"
      Loop_73 = 0
      while (Loop_73 < 2):
        $ 354 "bajar≔pose_add(get_actual_tcp_pose(), bajada_broca)"
        global bajar= pose_add ( get_actual_tcp_pose (), bajada_broca)
        $ 355 "bajar" "breakAfter"
        movel(bajar, a=0.005, v=0.001)
        $ 356 "subir≔pose_sub(get_actual_tcp_pose(), bajada_broca)"
        global subir= pose_sub ( get_actual_tcp_pose (), bajada_broca)
        $ 357 "subir" "breakAfter"
        movel(subir, a=0.01, v=0.005)
        $ 358 "bajada_broca≔pose_sub(bajada_broca, bajada)"
        global bajada_broca= pose_sub (bajada_broca, bajada)
        Loop_73 = Loop_73 + 1
      end
      $ 359 "Direction: Base Z+"
      global move_thread_flag_359=0
      thread move_thread_359():
        enter_critical
        move_thread_flag_359 = 1
        local towardsPos=calculate_point_to_move_towards(p[0.0,0.0,0.0,0.0,0.0,0.0], [0.0,0.0,1.0], 0.06)
        movel(towardsPos, a=0.035, v=0.03)
        move_thread_flag_359 = 2
        exit_critical
      end
      move_thread_flag_359 = 0
      move_thread_han_359 = run move_thread_359()
      while (True):
        sleep(1.0E-10)
        if (move_thread_flag_359 > 1):
          join move_thread_han_359
          $ 360 "Until (distance)"
          break
        end
        sync()
      end
      $ 361 "Set CO[1]=Apagar"
      set_configurable_digital_out(1, False)
      $ 362 "barreno_actual≔barreno_actual+1"
      global barreno_actual=barreno_actual+1
      $ 363 "Call Quitar_broca"
      Quitar_broca()
      $ 364 "Call Poner_broca"
      Poner_broca()
    end
    $ 365 "Popup: Linea1 con media Terminada!"
    popup("Linea1 con media Terminada!", "Mensaje", False, False, blocking=True)
    $ 366 "Linea2"
    $ 367 "Marcar_puntos"
    $ 368 "MoveL"
    $ 369 "Home2" "breakAfter"
    movel(Home2_p, a=0.5, v=0.1)
    $ 370 "Linea2_A" "breakAfter"
    movel(Linea2_A_p, a=0.5, v=0.1)
    $ 371 "Linea2_B" "breakAfter"
    movel(Linea2_B_p, a=0.5, v=0.1)
    $ 372 "Linea2_C" "breakAfter"
    movel(Linea2_C_p, a=0.5, v=0.1)
    $ 373 "Linea2_D" "breakAfter"
    movel(Linea2_D_p, a=0.5, v=0.1)
    $ 374 "Linea2_E" "breakAfter"
    movel(Linea2_E_p, a=0.5, v=0.1)
    $ 375 "Linea2_F" "breakAfter"
    movel(Linea2_F_p, a=0.5, v=0.1)
    $ 376 "AB"
    $ 377 "'desbaste_inicial'"
    # 'desbaste_inicial'
    $ 378 "bajada_broca≔p[0,0,-0.012,0,0,0]"
    global bajada_broca=p[0,0,-0.012,0,0,0]
    $ 379 "barrenos_menos1≔8"
    global barrenos_menos1=8
    $ 380 "barreno_actual≔0"
    global barreno_actual=0
    $ 381 "Loop barreno_actual≤barrenos_menos1"
    while (barreno_actual <= barrenos_menos1):
      $ 382 "Perforacion"
      $ 383 "MoveL"
      $ 384 "internos≔interpolate_pose(Linea2_A, Linea2_B, barreno_actual/barrenos_menos1)"
      global internos= interpolate_pose (Linea2_A_p, Linea2_B_p, barreno_actual/barrenos_menos1)
      $ 385 "internos" "breakAfter"
      movel(internos, a=0.5, v=0.1)
      $ 386 "'desbaste_inicial'"
      # 'desbaste_inicial'
      $ 387 "bajada_broca≔p[0,0,-0.012,0,0,0]"
      global bajada_broca=p[0,0,-0.012,0,0,0]
      $ 388 "bajada≔p[0,0,0.012,0,0,0]"
      global bajada=p[0,0,0.012,0,0,0]
      $ 389 "Direction: Base Z-"
      global move_thread_flag_389=0
      thread move_thread_389():
        enter_critical
        move_thread_flag_389 = 1
        local towardsPos=calculate_point_to_move_towards(p[0.0,0.0,0.0,0.0,0.0,0.0], [0.0,0.0,-1.0], 0.076)
        movel(towardsPos, a=0.015, v=0.015)
        move_thread_flag_389 = 2
        exit_critical
      end
      move_thread_flag_389 = 0
      move_thread_han_389 = run move_thread_389()
      while (True):
        sleep(1.0E-10)
        if (move_thread_flag_389 > 1):
          join move_thread_han_389
          $ 390 "Until (distance)"
          break
        end
        sync()
      end
      $ 391 "Popup: punto contacto alanzdo"
      popup("punto contacto alanzdo", "Mensaje", False, False, blocking=True)
      $ 392 "Direction: Base Z+"
      global move_thread_flag_392=0
      thread move_thread_392():
        enter_critical
        move_thread_flag_392 = 1
        local towardsPos=calculate_point_to_move_towards(p[0.0,0.0,0.0,0.0,0.0,0.0], [0.0,0.0,1.0], 0.002)
        movel(towardsPos, a=0.005, v=0.003)
        move_thread_flag_392 = 2
        exit_critical
      end
      move_thread_flag_392 = 0
      move_thread_han_392 = run move_thread_392()
      while (True):
        sleep(1.0E-10)
        if (move_thread_flag_392 > 1):
          join move_thread_han_392
          $ 393 "Until (distance)"
          break
        end
        sync()
      end
      $ 394 "Wait: 0.3"
      sleep(0.3)
      $ 395 "Set CO[1]=Encender"
      set_configurable_digital_out(1, True)
      $ 396 "Wait: 0.3"
      sleep(0.3)
      $ 397 "Loop 2 times"
      Loop_75 = 0
      while (Loop_75 < 2):
        $ 398 "bajar≔pose_add(get_actual_tcp_pose(), bajada_broca)"
        global bajar= pose_add ( get_actual_tcp_pose (), bajada_broca)
        $ 399 "bajar" "breakAfter"
        movel(bajar, a=0.005, v=0.001)
        $ 400 "subir≔pose_sub(get_actual_tcp_pose(), bajada_broca)"
        global subir= pose_sub ( get_actual_tcp_pose (), bajada_broca)
        $ 401 "subir" "breakAfter"
        movel(subir, a=0.01, v=0.005)
        $ 402 "bajada_broca≔pose_sub(bajada_broca, bajada)"
        global bajada_broca= pose_sub (bajada_broca, bajada)
        Loop_75 = Loop_75 + 1
      end
      $ 403 "Direction: Base Z+"
      global move_thread_flag_403=0
      thread move_thread_403():
        enter_critical
        move_thread_flag_403 = 1
        local towardsPos=calculate_point_to_move_towards(p[0.0,0.0,0.0,0.0,0.0,0.0], [0.0,0.0,1.0], 0.06)
        movel(towardsPos, a=0.035, v=0.03)
        move_thread_flag_403 = 2
        exit_critical
      end
      move_thread_flag_403 = 0
      move_thread_han_403 = run move_thread_403()
      while (True):
        sleep(1.0E-10)
        if (move_thread_flag_403 > 1):
          join move_thread_han_403
          $ 404 "Until (distance)"
          break
        end
        sync()
      end
      $ 405 "Set CO[1]=Apagar"
      set_configurable_digital_out(1, False)
      $ 406 "barreno_actual≔barreno_actual+1"
      global barreno_actual=barreno_actual+1
      $ 407 "Call Quitar_broca"
      Quitar_broca()
      $ 408 "Call Poner_broca"
      Poner_broca()
    end
    $ 409 "CD"
    $ 410 "'desbaste_inicial'"
    # 'desbaste_inicial'
    $ 411 "bajada_broca≔p[0,0,-0.012,0,0,0]"
    global bajada_broca=p[0,0,-0.012,0,0,0]
    $ 412 "barrenos_menos1≔8"
    global barrenos_menos1=8
    $ 413 "barreno_actual≔0"
    global barreno_actual=0
    $ 414 "Loop barreno_actual≤barrenos_menos1"
    while (barreno_actual <= barrenos_menos1):
      $ 415 "Perforacion"
      $ 416 "MoveL"
      $ 417 "internos≔interpolate_pose(Linea2_C, Linea2_D, barreno_actual/barrenos_menos1)"
      global internos= interpolate_pose (Linea2_C_p, Linea2_D_p, barreno_actual/barrenos_menos1)
      $ 418 "internos" "breakAfter"
      movel(internos, a=0.5, v=0.1)
      $ 419 "'desbaste_inicial'"
      # 'desbaste_inicial'
      $ 420 "bajada_broca≔p[0,0,-0.012,0,0,0]"
      global bajada_broca=p[0,0,-0.012,0,0,0]
      $ 421 "bajada≔p[0,0,0.012,0,0,0]"
      global bajada=p[0,0,0.012,0,0,0]
      $ 422 "Direction: Base Z-"
      global move_thread_flag_422=0
      thread move_thread_422():
        enter_critical
        move_thread_flag_422 = 1
        local towardsPos=calculate_point_to_move_towards(p[0.0,0.0,0.0,0.0,0.0,0.0], [0.0,0.0,-1.0], 0.076)
        movel(towardsPos, a=0.015, v=0.015)
        move_thread_flag_422 = 2
        exit_critical
      end
      move_thread_flag_422 = 0
      move_thread_han_422 = run move_thread_422()
      while (True):
        sleep(1.0E-10)
        if (move_thread_flag_422 > 1):
          join move_thread_han_422
          $ 423 "Until (distance)"
          break
        end
        sync()
      end
      $ 424 "Popup: punto contacto alanzdo"
      popup("punto contacto alanzdo", "Mensaje", False, False, blocking=True)
      $ 425 "Direction: Base Z+"
      global move_thread_flag_425=0
      thread move_thread_425():
        enter_critical
        move_thread_flag_425 = 1
        local towardsPos=calculate_point_to_move_towards(p[0.0,0.0,0.0,0.0,0.0,0.0], [0.0,0.0,1.0], 0.002)
        movel(towardsPos, a=0.005, v=0.003)
        move_thread_flag_425 = 2
        exit_critical
      end
      move_thread_flag_425 = 0
      move_thread_han_425 = run move_thread_425()
      while (True):
        sleep(1.0E-10)
        if (move_thread_flag_425 > 1):
          join move_thread_han_425
          $ 426 "Until (distance)"
          break
        end
        sync()
      end
      $ 427 "Wait: 0.3"
      sleep(0.3)
      $ 428 "Set CO[1]=Encender"
      set_configurable_digital_out(1, True)
      $ 429 "Wait: 0.3"
      sleep(0.3)
      $ 430 "Loop 2 times"
      Loop_78 = 0
      while (Loop_78 < 2):
        $ 431 "bajar≔pose_add(get_actual_tcp_pose(), bajada_broca)"
        global bajar= pose_add ( get_actual_tcp_pose (), bajada_broca)
        $ 432 "bajar" "breakAfter"
        movel(bajar, a=0.005, v=0.001)
        $ 433 "subir≔pose_sub(get_actual_tcp_pose(), bajada_broca)"
        global subir= pose_sub ( get_actual_tcp_pose (), bajada_broca)
        $ 434 "subir" "breakAfter"
        movel(subir, a=0.01, v=0.005)
        $ 435 "bajada_broca≔pose_sub(bajada_broca, bajada)"
        global bajada_broca= pose_sub (bajada_broca, bajada)
        Loop_78 = Loop_78 + 1
      end
      $ 436 "Direction: Base Z+"
      global move_thread_flag_436=0
      thread move_thread_436():
        enter_critical
        move_thread_flag_436 = 1
        local towardsPos=calculate_point_to_move_towards(p[0.0,0.0,0.0,0.0,0.0,0.0], [0.0,0.0,1.0], 0.06)
        movel(towardsPos, a=0.035, v=0.03)
        move_thread_flag_436 = 2
        exit_critical
      end
      move_thread_flag_436 = 0
      move_thread_han_436 = run move_thread_436()
      while (True):
        sleep(1.0E-10)
        if (move_thread_flag_436 > 1):
          join move_thread_han_436
          $ 437 "Until (distance)"
          break
        end
        sync()
      end
      $ 438 "Set CO[1]=Apagar"
      set_configurable_digital_out(1, False)
      $ 439 "barreno_actual≔barreno_actual+1"
      global barreno_actual=barreno_actual+1
      $ 440 "Call Quitar_broca"
      Quitar_broca()
      $ 441 "Call Poner_broca"
      Poner_broca()
    end
    $ 442 "EF"
    $ 443 "'desbaste_inicial'"
    # 'desbaste_inicial'
    $ 444 "bajada_broca≔p[0,0,-0.012,0,0,0]"
    global bajada_broca=p[0,0,-0.012,0,0,0]
    $ 445 "barrenos_menos1≔8"
    global barrenos_menos1=8
    $ 446 "barreno_actual≔0"
    global barreno_actual=0
    $ 447 "Loop barreno_actual≤barrenos_menos1"
    while (barreno_actual <= barrenos_menos1):
      $ 448 "Perforacion"
      $ 449 "MoveL"
      $ 450 "internos≔interpolate_pose(Linea2_E, Linea2_F, barreno_actual/barrenos_menos1)"
      global internos= interpolate_pose (Linea2_E_p, Linea2_F_p, barreno_actual/barrenos_menos1)
      $ 451 "internos" "breakAfter"
      movel(internos, a=0.5, v=0.1)
      $ 452 "'desbaste_inicial'"
      # 'desbaste_inicial'
      $ 453 "bajada_broca≔p[0,0,-0.012,0,0,0]"
      global bajada_broca=p[0,0,-0.012,0,0,0]
      $ 454 "bajada≔p[0,0,0.012,0,0,0]"
      global bajada=p[0,0,0.012,0,0,0]
      $ 455 "Direction: Base Z-"
      global move_thread_flag_455=0
      thread move_thread_455():
        enter_critical
        move_thread_flag_455 = 1
        local towardsPos=calculate_point_to_move_towards(p[0.0,0.0,0.0,0.0,0.0,0.0], [0.0,0.0,-1.0], 0.076)
        movel(towardsPos, a=0.015, v=0.015)
        move_thread_flag_455 = 2
        exit_critical
      end
      move_thread_flag_455 = 0
      move_thread_han_455 = run move_thread_455()
      while (True):
        sleep(1.0E-10)
        if (move_thread_flag_455 > 1):
          join move_thread_han_455
          $ 456 "Until (distance)"
          break
        end
        sync()
      end
      $ 457 "Popup: punto contacto alanzdo"
      popup("punto contacto alanzdo", "Mensaje", False, False, blocking=True)
      $ 458 "Direction: Base Z+"
      global move_thread_flag_458=0
      thread move_thread_458():
        enter_critical
        move_thread_flag_458 = 1
        local towardsPos=calculate_point_to_move_towards(p[0.0,0.0,0.0,0.0,0.0,0.0], [0.0,0.0,1.0], 0.002)
        movel(towardsPos, a=0.005, v=0.003)
        move_thread_flag_458 = 2
        exit_critical
      end
      move_thread_flag_458 = 0
      move_thread_han_458 = run move_thread_458()
      while (True):
        sleep(1.0E-10)
        if (move_thread_flag_458 > 1):
          join move_thread_han_458
          $ 459 "Until (distance)"
          break
        end
        sync()
      end
      $ 460 "Wait: 0.3"
      sleep(0.3)
      $ 461 "Set CO[1]=Encender"
      set_configurable_digital_out(1, True)
      $ 462 "Wait: 0.3"
      sleep(0.3)
      $ 463 "Loop 2 times"
      Loop_80 = 0
      while (Loop_80 < 2):
        $ 464 "bajar≔pose_add(get_actual_tcp_pose(), bajada_broca)"
        global bajar= pose_add ( get_actual_tcp_pose (), bajada_broca)
        $ 465 "bajar" "breakAfter"
        movel(bajar, a=0.005, v=0.001)
        $ 466 "subir≔pose_sub(get_actual_tcp_pose(), bajada_broca)"
        global subir= pose_sub ( get_actual_tcp_pose (), bajada_broca)
        $ 467 "subir" "breakAfter"
        movel(subir, a=0.01, v=0.005)
        $ 468 "bajada_broca≔pose_sub(bajada_broca, bajada)"
        global bajada_broca= pose_sub (bajada_broca, bajada)
        Loop_80 = Loop_80 + 1
      end
      $ 469 "Direction: Base Z+"
      global move_thread_flag_469=0
      thread move_thread_469():
        enter_critical
        move_thread_flag_469 = 1
        local towardsPos=calculate_point_to_move_towards(p[0.0,0.0,0.0,0.0,0.0,0.0], [0.0,0.0,1.0], 0.06)
        movel(towardsPos, a=0.035, v=0.03)
        move_thread_flag_469 = 2
        exit_critical
      end
      move_thread_flag_469 = 0
      move_thread_han_469 = run move_thread_469()
      while (True):
        sleep(1.0E-10)
        if (move_thread_flag_469 > 1):
          join move_thread_han_469
          $ 470 "Until (distance)"
          break
        end
        sync()
      end
      $ 471 "Set CO[1]=Apagar"
      set_configurable_digital_out(1, False)
      $ 472 "barreno_actual≔barreno_actual+1"
      global barreno_actual=barreno_actual+1
      $ 473 "If barreno_actual≥barrenos_menos1"
      if (barreno_actual >= barrenos_menos1):
        $ 474 "cambiar_broca≔ True "
        global cambiar_broca=  True
      end
      $ 475 "Call Quitar_broca"
      Quitar_broca()
      $ 476 "Call Poner_broca"
      Poner_broca()
    end
    $ 477 "Popup: Linea2 con media Terminada!"
    popup("Linea2 con media Terminada!", "Mensaje", False, False, blocking=True)
    $ 478 "Broca_3"
    $ 479 "Linea1"
    $ 480 "Marcar_puntos"
    $ 481 "MoveL"
    $ 482 "Home2" "breakAfter"
    movel(Home2_p, a=0.5, v=0.1)
    $ 483 "var"
    $ 484 "barrenos_hechos≔2"
    global barrenos_hechos=2
    $ 485 "eje7≔2"
    global eje7=2
    $ 486 "cambiar_broca≔ False "
    global cambiar_broca=  False
    $ 487 "iniciando_prog≔ False "
    global iniciando_prog=  False
    $ 488 "Linea1_A" "breakAfter"
    movel(Linea1_A_p, a=0.5, v=0.1)
    $ 489 "Linea1_B" "breakAfter"
    movel(Linea1_B_p, a=0.5, v=0.1)
    $ 490 "Linea1_C" "breakAfter"
    movel(Linea1_C_p, a=0.5, v=0.1)
    $ 491 "Linea1_D" "breakAfter"
    movel(Linea1_D_p, a=0.5, v=0.1)
    $ 492 "Linea1_E" "breakAfter"
    movel(Linea1_E_p, a=0.5, v=0.1)
    $ 493 "Linea1_F" "breakAfter"
    movel(Linea1_F_p, a=0.5, v=0.1)
    $ 494 "AB"
    $ 495 "'desbaste_inicial'"
    # 'desbaste_inicial'
    $ 496 "bajada_broca≔p[0,0,-0.012,0,0,0]"
    global bajada_broca=p[0,0,-0.012,0,0,0]
    $ 497 "barrenos_menos1≔8"
    global barrenos_menos1=8
    $ 498 "barreno_actual≔2"
    global barreno_actual=2
    $ 499 "Loop barreno_actual≤barrenos_menos1"
    while (barreno_actual <= barrenos_menos1):
      $ 500 "Perforacion"
      $ 501 "MoveL"
      $ 502 "internos≔interpolate_pose(Linea1_A, Linea1_B, barreno_actual/barrenos_menos1)"
      global internos= interpolate_pose (Linea1_A_p, Linea1_B_p, barreno_actual/barrenos_menos1)
      $ 503 "internos" "breakAfter"
      movel(internos, a=0.5, v=0.1)
      $ 504 "'desbaste_inicial'"
      # 'desbaste_inicial'
      $ 505 "bajada_broca≔p[0,0,-0.026,0,0,0]"
      global bajada_broca=p[0,0,-0.026,0,0,0]
      $ 506 "bajada≔p[0,0,0.026,0,0,0]"
      global bajada=p[0,0,0.026,0,0,0]
      $ 507 "Direction: Base Z-"
      global move_thread_flag_507=0
      thread move_thread_507():
        enter_critical
        move_thread_flag_507 = 1
        local towardsPos=calculate_point_to_move_towards(p[0.0,0.0,0.0,0.0,0.0,0.0], [0.0,0.0,-1.0], 0.08270000000000001)
        movel(towardsPos, a=0.015, v=0.015)
        move_thread_flag_507 = 2
        exit_critical
      end
      move_thread_flag_507 = 0
      move_thread_han_507 = run move_thread_507()
      while (True):
        sleep(1.0E-10)
        if (move_thread_flag_507 > 1):
          join move_thread_han_507
          $ 508 "Until (distance)"
          break
        end
        sync()
      end
      $ 509 "Popup: punto contacto alanzdo"
      popup("punto contacto alanzdo", "Mensaje", False, False, blocking=True)
      $ 510 "Direction: Base Z+"
      global move_thread_flag_510=0
      thread move_thread_510():
        enter_critical
        move_thread_flag_510 = 1
        local towardsPos=calculate_point_to_move_towards(p[0.0,0.0,0.0,0.0,0.0,0.0], [0.0,0.0,1.0], 0.002)
        movel(towardsPos, a=0.005, v=0.003)
        move_thread_flag_510 = 2
        exit_critical
      end
      move_thread_flag_510 = 0
      move_thread_han_510 = run move_thread_510()
      while (True):
        sleep(1.0E-10)
        if (move_thread_flag_510 > 1):
          join move_thread_han_510
          $ 511 "Until (distance)"
          break
        end
        sync()
      end
      $ 512 "Wait: 0.3"
      sleep(0.3)
      $ 513 "Set CO[1]=Encender"
      set_configurable_digital_out(1, True)
      $ 514 "Wait: 0.3"
      sleep(0.3)
      $ 515 "Loop 1 times"
      Loop_82 = 0
      while (Loop_82 < 1):
        $ 516 "bajar≔pose_add(get_actual_tcp_pose(), bajada_broca)"
        global bajar= pose_add ( get_actual_tcp_pose (), bajada_broca)
        $ 517 "bajar" "breakAfter"
        movel(bajar, a=0.005, v=0.001)
        $ 518 "subir≔pose_sub(get_actual_tcp_pose(), bajada_broca)"
        global subir= pose_sub ( get_actual_tcp_pose (), bajada_broca)
        $ 519 "subir" "breakAfter"
        movel(subir, a=0.01, v=0.005)
        $ 520 "bajada_broca≔pose_sub(bajada_broca, bajada)"
        global bajada_broca= pose_sub (bajada_broca, bajada)
        Loop_82 = Loop_82 + 1
      end
      $ 521 "Direction: Base Z+"
      global move_thread_flag_521=0
      thread move_thread_521():
        enter_critical
        move_thread_flag_521 = 1
        local towardsPos=calculate_point_to_move_towards(p[0.0,0.0,0.0,0.0,0.0,0.0], [0.0,0.0,1.0], 0.06)
        movel(towardsPos, a=0.035, v=0.03)
        move_thread_flag_521 = 2
        exit_critical
      end
      move_thread_flag_521 = 0
      move_thread_han_521 = run move_thread_521()
      while (True):
        sleep(1.0E-10)
        if (move_thread_flag_521 > 1):
          join move_thread_han_521
          $ 522 "Until (distance)"
          break
        end
        sync()
      end
      $ 523 "Set CO[1]=Apagar"
      set_configurable_digital_out(1, False)
      $ 524 "barreno_actual≔barreno_actual+1"
      global barreno_actual=barreno_actual+1
      $ 525 "Call Quitar_broca"
      Quitar_broca()
      $ 526 "Call Poner_broca"
      Poner_broca()
    end
    $ 527 "CD"
    $ 528 "'desbaste_inicial'"
    # 'desbaste_inicial'
    $ 529 "bajada_broca≔p[0,0,-0.012,0,0,0]"
    global bajada_broca=p[0,0,-0.012,0,0,0]
    $ 530 "barrenos_menos1≔8"
    global barrenos_menos1=8
    $ 531 "barreno_actual≔5"
    global barreno_actual=5
    $ 532 "Loop barreno_actual≤barrenos_menos1"
    while (barreno_actual <= barrenos_menos1):
      $ 533 "Perforacion"
      $ 534 "MoveL"
      $ 535 "internos≔interpolate_pose(Linea1_C, Linea1_D, barreno_actual/barrenos_menos1)"
      global internos= interpolate_pose (Linea1_C_p, Linea1_D_p, barreno_actual/barrenos_menos1)
      $ 536 "internos" "breakAfter"
      movel(internos, a=0.5, v=0.1)
      $ 537 "'desbaste_inicial'"
      # 'desbaste_inicial'
      $ 538 "bajada_broca≔p[0,0,-0.026,0,0,0]"
      global bajada_broca=p[0,0,-0.026,0,0,0]
      $ 539 "bajada≔p[0,0,0.026,0,0,0]"
      global bajada=p[0,0,0.026,0,0,0]
      $ 540 "Direction: Base Z-"
      global move_thread_flag_540=0
      thread move_thread_540():
        enter_critical
        move_thread_flag_540 = 1
        local towardsPos=calculate_point_to_move_towards(p[0.0,0.0,0.0,0.0,0.0,0.0], [0.0,0.0,-1.0], 0.08270000000000001)
        movel(towardsPos, a=0.015, v=0.015)
        move_thread_flag_540 = 2
        exit_critical
      end
      move_thread_flag_540 = 0
      move_thread_han_540 = run move_thread_540()
      while (True):
        sleep(1.0E-10)
        if (move_thread_flag_540 > 1):
          join move_thread_han_540
          $ 541 "Until (distance)"
          break
        end
        sync()
      end
      $ 542 "Popup: punto contacto alanzdo"
      popup("punto contacto alanzdo", "Mensaje", False, False, blocking=True)
      $ 543 "Direction: Base Z+"
      global move_thread_flag_543=0
      thread move_thread_543():
        enter_critical
        move_thread_flag_543 = 1
        local towardsPos=calculate_point_to_move_towards(p[0.0,0.0,0.0,0.0,0.0,0.0], [0.0,0.0,1.0], 0.002)
        movel(towardsPos, a=0.005, v=0.003)
        move_thread_flag_543 = 2
        exit_critical
      end
      move_thread_flag_543 = 0
      move_thread_han_543 = run move_thread_543()
      while (True):
        sleep(1.0E-10)
        if (move_thread_flag_543 > 1):
          join move_thread_han_543
          $ 544 "Until (distance)"
          break
        end
        sync()
